ABB RobotStudio station: solution_2_AI.rspag

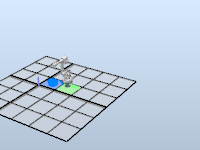
--- station ---
Station test (saved by RobotStudio 20.4.9280.0)
Controller Controller_IRB2600_12_165_C, task T_ROB1: task frame (RAPID world) sits at (1280, 730, 300) mm, rotated rx 0 ry 0 rz -90 deg in the station
Controller Controller_IRB2600_12_165_C
  mechanical unit ROB_1: IRB2600_12_165_C_01_2, 6 joints, base frame (0, 0, 0) mm
Layout (positions relative to the parent item):
  - 机器人区 [part] at (1507.5, 502.5, 0) mm
  - 方块产生区 [part]
  - 删行控制器 [smart component]
      signals: DI Rows_Delete
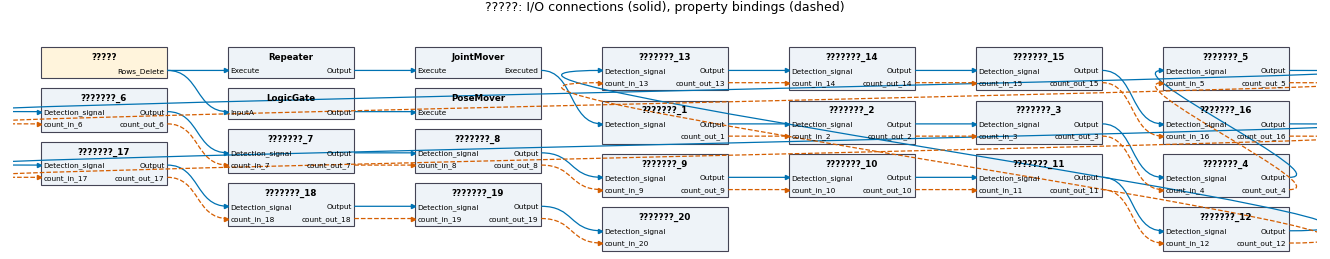
      connections:
        Repeater.Output -> JointMover.Execute
        删行控制器.Rows_Delete -> Repeater.Execute
        删行控制器.Rows_Delete -> LogicGate.InputA
        LogicGate.Output -> PoseMover.Execute
        JointMover.Executed -> 满行检测与下坠_1.Detection_signal
        满行检测与下坠_1.Output -> 满行检测与下坠_2.Detection_signal
        满行检测与下坠_2.Output -> 满行检测与下坠_3.Detection_signal
        满行检测与下坠_3.Output -> 满行检测与下坠_4.Detection_signal
        满行检测与下坠_4.Output -> 满行检测与下坠_5.Detection_signal
        满行检测与下坠_5.Output -> 满行检测与下坠_6.Detection_signal
        满行检测与下坠_6.Output -> 满行检测与下坠_7.Detection_signal
        满行检测与下坠_7.Output -> 满行检测与下坠_8.Detection_signal
        满行检测与下坠_10.Output -> 满行检测与下坠_11.Detection_signal
        满行检测与下坠_11.Output -> 满行检测与下坠_12.Detection_signal
        满行检测与下坠_12.Output -> 满行检测与下坠_13.Detection_signal
        满行检测与下坠_13.Output -> 满行检测与下坠_14.Detection_signal
        满行检测与下坠_14.Output -> 满行检测与下坠_15.Detection_signal
        满行检测与下坠_15.Output -> 满行检测与下坠_16.Detection_signal
        满行检测与下坠_16.Output -> 满行检测与下坠_17.Detection_signal
        满行检测与下坠_17.Output -> 满行检测与下坠_18.Detection_signal
        满行检测与下坠_18.Output -> 满行检测与下坠_19.Detection_signal
        满行检测与下坠_19.Output -> 满行检测与下坠_20.Detection_signal
        满行检测与下坠_8.Output -> 满行检测与下坠_9.Detection_signal
        满行检测与下坠_9.Output -> 满行检测与下坠_10.Detection_signal
        满行检测与下坠_1.count_out_1 => 满行检测与下坠_2.count_in_2
        满行检测与下坠_2.count_out_2 => 满行检测与下坠_3.count_in_3
        满行检测与下坠_3.count_out_3 => 满行检测与下坠_4.count_in_4
        满行检测与下坠_4.count_out_4 => 满行检测与下坠_5.count_in_5
        满行检测与下坠_5.count_out_5 => 满行检测与下坠_6.count_in_6
        满行检测与下坠_6.count_out_6 => 满行检测与下坠_7.count_in_7
        满行检测与下坠_7.count_out_7 => 满行检测与下坠_8.count_in_8
        满行检测与下坠_8.count_out_8 => 满行检测与下坠_9.count_in_9
        满行检测与下坠_9.count_out_9 => 满行检测与下坠_10.count_in_10
        满行检测与下坠_10.count_out_10 => 满行检测与下坠_11.count_in_11
        满行检测与下坠_11.count_out_11 => 满行检测与下坠_12.count_in_12
        满行检测与下坠_12.count_out_12 => 满行检测与下坠_13.count_in_13
        满行检测与下坠_13.count_out_13 => 满行检测与下坠_14.count_in_14
        满行检测与下坠_14.count_out_14 => 满行检测与下坠_15.count_in_15
        满行检测与下坠_15.count_out_15 => 满行检测与下坠_16.count_in_16
        满行检测与下坠_16.count_out_16 => 满行检测与下坠_17.count_in_17
        满行检测与下坠_17.count_out_17 => 满行检测与下坠_18.count_in_18
        满行检测与下坠_18.count_out_18 => 满行检测与下坠_19.count_in_19
        满行检测与下坠_19.count_out_19 => 满行检测与下坠_20.count_in_20
    - 扫描式传感器 [mechanism] at (0, -50, 0) mm; joint values [0] (rad or m)
        links: L1, L2
    - JointMover [smart component, from Components\JointMover.rslib]
        properties: Mechanism=扫描式传感器; Relative=true; Duration=0; J1=0.1
    - Repeater [smart component, from Components\Repeater.rslib]
        properties: Count=10
    - PoseMover [smart component, from Components\PoseMover.rslib]
        properties: Mechanism=扫描式传感器; Pose=0; Duration=0
    - 满行检测与下坠_1 [smart component]
        properties: count_in_1=0; count_out_1=0
        signals: DI Detection_signal, DO Output
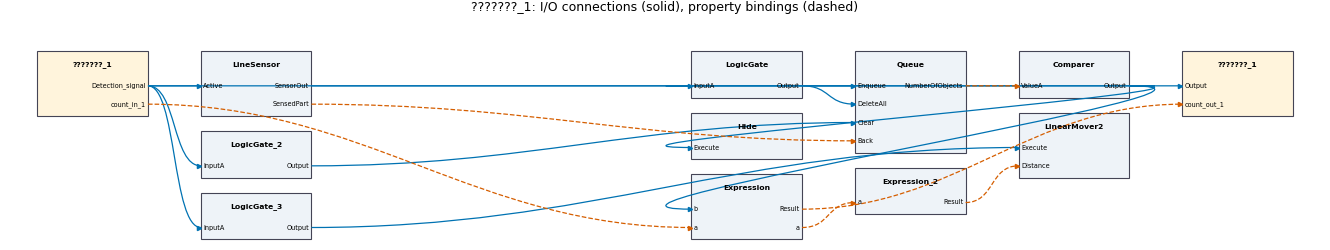
        connections:
          满行检测与下坠_1.Detection_signal -> LineSensor.Active
          LineSensor.SensorOut -> Queue.Enqueue
          Comparer.Output -> LogicGate.InputA
          LogicGate.Output -> Queue.DeleteAll
          Comparer.Output -> Hide.Execute
          LogicGate_2.Output -> Queue.Clear
          满行检测与下坠_1.Detection_signal -> LogicGate_2.InputA
          Comparer.Output -> Expression.b
          满行检测与下坠_1.Detection_signal -> LogicGate_3.InputA
          LogicGate_3.Output -> LinearMover2.Execute
          满行检测与下坠_1.Detection_signal -> 满行检测与下坠_1.Output
          LineSensor.SensedPart => Queue.Back
          Queue.NumberOfObjects => Comparer.ValueA
          满行检测与下坠_1.count_in_1 => Expression.a
          Expression.Result => 满行检测与下坠_1.count_out_1
          Expression.a => Expression_2.a
          Expression_2.Result => LinearMover2.Distance
      - LineSensor [smart component, from Components\LineSensor.rslib] at (0, 0, 40) mm
          properties: Start=[2.06 -0.045 0.01]; End=[2.13 -0.045 0.01]; Radius=0.002; SensedPart=(none); SensedPoint=[0 0 0]
        - _sensorPart_ [part]
      - Queue [smart component, from Components\Queue.rslib]
          properties: Back=(none); Front=(none); Queue=; NumberOfObjects=0
      - Comparer [smart component, from Components\Comparer.rslib]
          properties: ValueA=0; Operator===; ValueB=10
      - LogicGate [smart component, from Components\LogicGate.rslib]
          properties: Operator=NOP; Delay=0.6
      - Hide [smart component, from Components\Hide.rslib]
          properties: Object=Queue
      - LogicGate_2 [smart component, from Components\LogicGate.rslib]
          properties: Operator=NOP; Delay=0.7
      - Expression [smart component, from Components\Expression.rslib]
          properties: Expression=a+b; Result=0; a=0; b=0
      - LinearMover2 [smart component, from Components\LinearMover2.rslib]
          properties: Object=Queue; Direction=[0 0 -0.001]; Distance=0; Duration=0.5; Reference=Global; ReferenceObject=(none)
      - LogicGate_3 [smart component, from Components\LogicGate.rslib]
          properties: Operator=NOP; Delay=0.1
      - Expression_2 [smart component, from Components\Expression.rslib]
          properties: Expression=a/10; Result=0; a=0
    - LogicGate [smart component, from Components\LogicGate.rslib]
        properties: Operator=NOP; Delay=0.024
    - 满行检测与下坠_2 [smart component] at (0, 0, 100) mm
        properties: count_in_1=0; count_out_1=0; count_in_2=0; count_out_2=0
        signals: DI Detection_signal, DO Output
        connections:
          满行检测与下坠_2.Detection_signal -> LineSensor.Active
          LineSensor.SensorOut -> Queue.Enqueue
          Comparer.Output -> LogicGate.InputA
          LogicGate.Output -> Queue.DeleteAll
          Comparer.Output -> Hide.Execute
          LogicGate_2.Output -> Queue.Clear
          满行检测与下坠_2.Detection_signal -> LogicGate_2.InputA
          Comparer.Output -> Expression.b
          满行检测与下坠_2.Detection_signal -> LogicGate_3.InputA
          LogicGate_3.Output -> LinearMover2.Execute
          满行检测与下坠_2.Detection_signal -> 满行检测与下坠_2.Output
          LineSensor.SensedPart => Queue.Back
          Queue.NumberOfObjects => Comparer.ValueA
          Expression.a => Expression_2.a
          Expression_2.Result => LinearMover2.Distance
          满行检测与下坠_2.count_in_2 => Expression.a
          Expression.Result => 满行检测与下坠_2.count_out_2
      - LineSensor [smart component, from Components\LineSensor.rslib] at (0, 0, 40) mm
          properties: Start=[2.06 -0.045 0.01]; End=[2.13 -0.045 0.01]; Radius=0.002; SensedPart=(none); SensedPoint=[0 0 0]
        - _sensorPart_ [part]
      - Queue [smart component, from Components\Queue.rslib]
          properties: Back=(none); Front=(none); Queue=; NumberOfObjects=0
      - Comparer [smart component, from Components\Comparer.rslib]
          properties: ValueA=0; Operator===; ValueB=10
      - LogicGate [smart component, from Components\LogicGate.rslib]
          properties: Operator=NOP; Delay=0.6
      - Hide [smart component, from Components\Hide.rslib]
          properties: Object=Queue
      - LogicGate_2 [smart component, from Components\LogicGate.rslib]
          properties: Operator=NOP; Delay=0.7
      - Expression [smart component, from Components\Expression.rslib]
          properties: Expression=a+b; Result=0; a=0; b=0
      - LinearMover2 [smart component, from Components\LinearMover2.rslib]
          properties: Object=Queue; Direction=[0 0 -0.001]; Distance=0; Duration=0.5; Reference=Global; ReferenceObject=(none)
      - LogicGate_3 [smart component, from Components\LogicGate.rslib]
          properties: Operator=NOP; Delay=0.1
      - Expression_2 [smart component, from Components\Expression.rslib]
          properties: Expression=a/10; Result=0; a=0
    - 满行检测与下坠_3 [smart component] at (0, 0, 200) mm
        properties: count_in_1=0; count_out_1=0; count_in_3=0; count_out_3=0
        signals: DI Detection_signal, DO Output
        connections:
          满行检测与下坠_3.Detection_signal -> LineSensor.Active
          LineSensor.SensorOut -> Queue.Enqueue
          Comparer.Output -> LogicGate.InputA
          LogicGate.Output -> Queue.DeleteAll
          Comparer.Output -> Hide.Execute
          LogicGate_2.Output -> Queue.Clear
          满行检测与下坠_3.Detection_signal -> LogicGate_2.InputA
          Comparer.Output -> Expression.b
          满行检测与下坠_3.Detection_signal -> LogicGate_3.InputA
          LogicGate_3.Output -> LinearMover2.Execute
          满行检测与下坠_3.Detection_signal -> 满行检测与下坠_3.Output
          LineSensor.SensedPart => Queue.Back
          Queue.NumberOfObjects => Comparer.ValueA
          Expression.a => Expression_2.a
          Expression_2.Result => LinearMover2.Distance
          满行检测与下坠_3.count_in_3 => Expression.a
          Expression.Result => 满行检测与下坠_3.count_out_3
      - LineSensor [smart component, from Components\LineSensor.rslib] at (0, 0, 40) mm
          properties: Start=[2.06 -0.045 0.01]; End=[2.13 -0.045 0.01]; Radius=0.002; SensedPart=(none); SensedPoint=[0 0 0]
        - _sensorPart_ [part]
      - Queue [smart component, from Components\Queue.rslib]
          properties: Back=(none); Front=(none); Queue=; NumberOfObjects=0
      - Comparer [smart component, from Components\Comparer.rslib]
          properties: ValueA=0; Operator===; ValueB=10
      - LogicGate [smart component, from Components\LogicGate.rslib]
          properties: Operator=NOP; Delay=0.6
      - Hide [smart component, from Components\Hide.rslib]
          properties: Object=Queue
      - LogicGate_2 [smart component, from Components\LogicGate.rslib]
          properties: Operator=NOP; Delay=0.7
      - Expression [smart component, from Components\Expression.rslib]
          properties: Expression=a+b; Result=0; a=0; b=0
      - LinearMover2 [smart component, from Components\LinearMover2.rslib]
          properties: Object=Queue; Direction=[0 0 -0.001]; Distance=0; Duration=0.5; Reference=Global; ReferenceObject=(none)
      - LogicGate_3 [smart component, from Components\LogicGate.rslib]
          properties: Operator=NOP; Delay=0.1
      - Expression_2 [smart component, from Components\Expression.rslib]
          properties: Expression=a/10; Result=0; a=0
    - 满行检测与下坠_4 [smart component] at (0, 0, 300) mm
        properties: count_in_1=0; count_out_1=0; count_in_4=0; count_out_4=0
        signals: DI Detection_signal, DO Output
        connections:
          满行检测与下坠_4.Detection_signal -> LineSensor.Active
          LineSensor.SensorOut -> Queue.Enqueue
          Comparer.Output -> LogicGate.InputA
          LogicGate.Output -> Queue.DeleteAll
          Comparer.Output -> Hide.Execute
          LogicGate_2.Output -> Queue.Clear
          满行检测与下坠_4.Detection_signal -> LogicGate_2.InputA
          Comparer.Output -> Expression.b
          满行检测与下坠_4.Detection_signal -> LogicGate_3.InputA
          LogicGate_3.Output -> LinearMover2.Execute
          满行检测与下坠_4.Detection_signal -> 满行检测与下坠_4.Output
          LineSensor.SensedPart => Queue.Back
          Queue.NumberOfObjects => Comparer.ValueA
          Expression.a => Expression_2.a
          Expression_2.Result => LinearMover2.Distance
          满行检测与下坠_4.count_in_4 => Expression.a
          Expression.Result => 满行检测与下坠_4.count_out_4
      - LineSensor [smart component, from Components\LineSensor.rslib] at (0, 0, 40) mm
          properties: Start=[2.06 -0.045 0.01]; End=[2.13 -0.045 0.01]; Radius=0.002; SensedPart=(none); SensedPoint=[0 0 0]
        - _sensorPart_ [part]
      - Queue [smart component, from Components\Queue.rslib]
          properties: Back=(none); Front=(none); Queue=; NumberOfObjects=0
      - Comparer [smart component, from Components\Comparer.rslib]
          properties: ValueA=0; Operator===; ValueB=10
      - LogicGate [smart component, from Components\LogicGate.rslib]
          properties: Operator=NOP; Delay=0.6
      - Hide [smart component, from Components\Hide.rslib]
          properties: Object=Queue
      - LogicGate_2 [smart component, from Components\LogicGate.rslib]
          properties: Operator=NOP; Delay=0.7
      - Expression [smart component, from Components\Expression.rslib]
          properties: Expression=a+b; Result=0; a=0; b=0
      - LinearMover2 [smart component, from Components\LinearMover2.rslib]
          properties: Object=Queue; Direction=[0 0 -0.001]; Distance=0; Duration=0.5; Reference=Global; ReferenceObject=(none)
      - LogicGate_3 [smart component, from Components\LogicGate.rslib]
          properties: Operator=NOP; Delay=0.1
      - Expression_2 [smart component, from Components\Expression.rslib]
          properties: Expression=a/10; Result=0; a=0
    - 满行检测与下坠_5 [smart component] at (0, 0, 400) mm
        properties: count_in_1=0; count_out_1=0; count_in_5=0; count_out_5=0
        signals: DI Detection_signal, DO Output
        connections:
          满行检测与下坠_5.Detection_signal -> LineSensor.Active
          LineSensor.SensorOut -> Queue.Enqueue
          Comparer.Output -> LogicGate.InputA
          LogicGate.Output -> Queue.DeleteAll
          Comparer.Output -> Hide.Execute
          LogicGate_2.Output -> Queue.Clear
          满行检测与下坠_5.Detection_signal -> LogicGate_2.InputA
          Comparer.Output -> Expression.b
          满行检测与下坠_5.Detection_signal -> LogicGate_3.InputA
          LogicGate_3.Output -> LinearMover2.Execute
          满行检测与下坠_5.Detection_signal -> 满行检测与下坠_5.Output
          LineSensor.SensedPart => Queue.Back
          Queue.NumberOfObjects => Comparer.ValueA
          Expression.a => Expression_2.a
          Expression_2.Result => LinearMover2.Distance
          满行检测与下坠_5.count_in_5 => Expression.a
          Expression.Result => 满行检测与下坠_5.count_out_5
      - LineSensor [smart component, from Components\LineSensor.rslib] at (0, 0, 40) mm
          properties: Start=[2.06 -0.045 0.01]; End=[2.13 -0.045 0.01]; Radius=0.002; SensedPart=(none); SensedPoint=[0 0 0]
        - _sensorPart_ [part]
      - Queue [smart component, from Components\Queue.rslib]
          properties: Back=(none); Front=(none); Queue=; NumberOfObjects=0
      - Comparer [smart component, from Components\Comparer.rslib]
          properties: ValueA=0; Operator===; ValueB=10
      - LogicGate [smart component, from Components\LogicGate.rslib]
          properties: Operator=NOP; Delay=0.6
      - Hide [smart component, from Components\Hide.rslib]
          properties: Object=Queue
      - LogicGate_2 [smart component, from Components\LogicGate.rslib]
          properties: Operator=NOP; Delay=0.7
      - Expression [smart component, from Components\Expression.rslib]
          properties: Expression=a+b; Result=0; a=0; b=0
      - LinearMover2 [smart component, from Components\LinearMover2.rslib]
          properties: Object=Queue; Direction=[0 0 -0.001]; Distance=0; Duration=0.5; Reference=Global; ReferenceObject=(none)
      - LogicGate_3 [smart component, from Components\LogicGate.rslib]
          properties: Operator=NOP; Delay=0.1
      - Expression_2 [smart component, from Components\Expression.rslib]
          properties: Expression=a/10; Result=0; a=0
    - 满行检测与下坠_6 [smart component] at (0, 0, 500) mm
        properties: count_in_1=0; count_out_1=0; count_in_6=0; count_out_6=0
        signals: DI Detection_signal, DO Output
        connections:
          满行检测与下坠_6.Detection_signal -> LineSensor.Active
          LineSensor.SensorOut -> Queue.Enqueue
          Comparer.Output -> LogicGate.InputA
          LogicGate.Output -> Queue.DeleteAll
          Comparer.Output -> Hide.Execute
          LogicGate_2.Output -> Queue.Clear
          满行检测与下坠_6.Detection_signal -> LogicGate_2.InputA
          Comparer.Output -> Expression.b
          满行检测与下坠_6.Detection_signal -> LogicGate_3.InputA
          LogicGate_3.Output -> LinearMover2.Execute
          满行检测与下坠_6.Detection_signal -> 满行检测与下坠_6.Output
          LineSensor.SensedPart => Queue.Back
          Queue.NumberOfObjects => Comparer.ValueA
          Expression.a => Expression_2.a
          Expression_2.Result => LinearMover2.Distance
          满行检测与下坠_6.count_in_6 => Expression.a
          Expression.Result => 满行检测与下坠_6.count_out_6
      - LineSensor [smart component, from Components\LineSensor.rslib] at (0, 0, 40) mm
          properties: Start=[2.06 -0.045 0.01]; End=[2.13 -0.045 0.01]; Radius=0.002; SensedPart=(none); SensedPoint=[0 0 0]
        - _sensorPart_ [part]
      - Queue [smart component, from Components\Queue.rslib]
          properties: Back=(none); Front=(none); Queue=; NumberOfObjects=0
      - Comparer [smart component, from Components\Comparer.rslib]
          properties: ValueA=0; Operator===; ValueB=10
      - LogicGate [smart component, from Components\LogicGate.rslib]
          properties: Operator=NOP; Delay=0.6
      - Hide [smart component, from Components\Hide.rslib]
          properties: Object=Queue
      - LogicGate_2 [smart component, from Components\LogicGate.rslib]
          properties: Operator=NOP; Delay=0.7
      - Expression [smart component, from Components\Expression.rslib]
          properties: Expression=a+b; Result=0; a=0; b=0
      - LinearMover2 [smart component, from Components\LinearMover2.rslib]
          properties: Object=Queue; Direction=[0 0 -0.001]; Distance=0; Duration=0.5; Reference=Global; ReferenceObject=(none)
      - LogicGate_3 [smart component, from Components\LogicGate.rslib]
          properties: Operator=NOP; Delay=0.1
      - Expression_2 [smart component, from Components\Expression.rslib]
          properties: Expression=a/10; Result=0; a=0
    - 满行检测与下坠_7 [smart component] at (0, 0, 600) mm
        properties: count_in_1=0; count_out_1=0; count_in_7=0; count_out_8=0; count_out_7=0
        signals: DI Detection_signal, DO Output
        connections:
          满行检测与下坠_7.Detection_signal -> LineSensor.Active
          LineSensor.SensorOut -> Queue.Enqueue
          Comparer.Output -> LogicGate.InputA
          LogicGate.Output -> Queue.DeleteAll
          Comparer.Output -> Hide.Execute
          LogicGate_2.Output -> Queue.Clear
          满行检测与下坠_7.Detection_signal -> LogicGate_2.InputA
          Comparer.Output -> Expression.b
          满行检测与下坠_7.Detection_signal -> LogicGate_3.InputA
          LogicGate_3.Output -> LinearMover2.Execute
          满行检测与下坠_7.Detection_signal -> 满行检测与下坠_7.Output
          LineSensor.SensedPart => Queue.Back
          Queue.NumberOfObjects => Comparer.ValueA
          Expression.a => Expression_2.a
          Expression_2.Result => LinearMover2.Distance
          满行检测与下坠_7.count_in_7 => Expression.a
          Expression.Result => 满行检测与下坠_7.count_out_7
      - LineSensor [smart component, from Components\LineSensor.rslib] at (0, 0, 40) mm
          properties: Start=[2.06 -0.045 0.01]; End=[2.13 -0.045 0.01]; Radius=0.002; SensedPart=(none); SensedPoint=[0 0 0]
        - _sensorPart_ [part]
      - Queue [smart component, from Components\Queue.rslib]
          properties: Back=(none); Front=(none); Queue=; NumberOfObjects=0
      - Comparer [smart component, from Components\Comparer.rslib]
          properties: ValueA=0; Operator===; ValueB=10
      - LogicGate [smart component, from Components\LogicGate.rslib]
          properties: Operator=NOP; Delay=0.6
      - Hide [smart component, from Components\Hide.rslib]
          properties: Object=Queue
      - LogicGate_2 [smart component, from Components\LogicGate.rslib]
          properties: Operator=NOP; Delay=0.7
      - Expression [smart component, from Components\Expression.rslib]
          properties: Expression=a+b; Result=0; a=0; b=0
      - LinearMover2 [smart component, from Components\LinearMover2.rslib]
          properties: Object=Queue; Direction=[0 0 -0.001]; Distance=0; Duration=0.5; Reference=Global; ReferenceObject=(none)
      - LogicGate_3 [smart component, from Components\LogicGate.rslib]
          properties: Operator=NOP; Delay=0.1
      - Expression_2 [smart component, from Components\Expression.rslib]
          properties: Expression=a/10; Result=0; a=0
    - 满行检测与下坠_8 [smart component] at (0, 0, 700) mm
        properties: count_in_1=0; count_out_1=0; count_in_8=0; count_out_8=0
        signals: DI Detection_signal, DO Output
        connections:
          满行检测与下坠_8.Detection_signal -> LineSensor.Active
          LineSensor.SensorOut -> Queue.Enqueue
          Comparer.Output -> LogicGate.InputA
          LogicGate.Output -> Queue.DeleteAll
          Comparer.Output -> Hide.Execute
          LogicGate_2.Output -> Queue.Clear
          满行检测与下坠_8.Detection_signal -> LogicGate_2.InputA
          Comparer.Output -> Expression.b
          满行检测与下坠_8.Detection_signal -> LogicGate_3.InputA
          LogicGate_3.Output -> LinearMover2.Execute
          满行检测与下坠_8.Detection_signal -> 满行检测与下坠_8.Output
          LineSensor.SensedPart => Queue.Back
          Queue.NumberOfObjects => Comparer.ValueA
          Expression.a => Expression_2.a
          Expression_2.Result => LinearMover2.Distance
          满行检测与下坠_8.count_in_8 => Expression.a
          Expression.Result => 满行检测与下坠_8.count_out_8
      - LineSensor [smart component, from Components\LineSensor.rslib] at (0, 0, 40) mm
          properties: Start=[2.06 -0.045 0.01]; End=[2.13 -0.045 0.01]; Radius=0.002; SensedPart=(none); SensedPoint=[0 0 0]
        - _sensorPart_ [part]
      - Queue [smart component, from Components\Queue.rslib]
          properties: Back=(none); Front=(none); Queue=; NumberOfObjects=0
      - Comparer [smart component, from Components\Comparer.rslib]
          properties: ValueA=0; Operator===; ValueB=10
      - LogicGate [smart component, from Components\LogicGate.rslib]
          properties: Operator=NOP; Delay=0.6
      - Hide [smart component, from Components\Hide.rslib]
          properties: Object=Queue
      - LogicGate_2 [smart component, from Components\LogicGate.rslib]
          properties: Operator=NOP; Delay=0.7
      - Expression [smart component, from Components\Expression.rslib]
          properties: Expression=a+b; Result=0; a=0; b=0
      - LinearMover2 [smart component, from Components\LinearMover2.rslib]
          properties: Object=Queue; Direction=[0 0 -0.001]; Distance=0; Duration=0.5; Reference=Global; ReferenceObject=(none)
      - LogicGate_3 [smart component, from Components\LogicGate.rslib]
          properties: Operator=NOP; Delay=0.1
      - Expression_2 [smart component, from Components\Expression.rslib]
          properties: Expression=a/10; Result=0; a=0
    - 满行检测与下坠_9 [smart component] at (0, 0, 800) mm
        properties: count_in_1=0; count_out_1=0; count_in_9=0; count_out_9=0
        signals: DI Detection_signal, DO Output
        connections:
          满行检测与下坠_9.Detection_signal -> LineSensor.Active
          LineSensor.SensorOut -> Queue.Enqueue
          Comparer.Output -> LogicGate.InputA
          LogicGate.Output -> Queue.DeleteAll
          Comparer.Output -> Hide.Execute
          LogicGate_2.Output -> Queue.Clear
          满行检测与下坠_9.Detection_signal -> LogicGate_2.InputA
          Comparer.Output -> Expression.b
          满行检测与下坠_9.Detection_signal -> LogicGate_3.InputA
          LogicGate_3.Output -> LinearMover2.Execute
          满行检测与下坠_9.Detection_signal -> 满行检测与下坠_9.Output
          LineSensor.SensedPart => Queue.Back
          Queue.NumberOfObjects => Comparer.ValueA
          Expression.a => Expression_2.a
          Expression_2.Result => LinearMover2.Distance
          满行检测与下坠_9.count_in_9 => Expression.a
          Expression.Result => 满行检测与下坠_9.count_out_9
      - LineSensor [smart component, from Components\LineSensor.rslib] at (0, 0, 40) mm
          properties: Start=[2.06 -0.045 0.01]; End=[2.13 -0.045 0.01]; Radius=0.002; SensedPart=(none); SensedPoint=[0 0 0]
        - _sensorPart_ [part]
      - Queue [smart component, from Components\Queue.rslib]
          properties: Back=(none); Front=(none); Queue=; NumberOfObjects=0
      - Comparer [smart component, from Components\Comparer.rslib]
          properties: ValueA=0; Operator===; ValueB=10
      - LogicGate [smart component, from Components\LogicGate.rslib]
          properties: Operator=NOP; Delay=0.6
      - Hide [smart component, from Components\Hide.rslib]
          properties: Object=Queue
      - LogicGate_2 [smart component, from Components\LogicGate.rslib]
          properties: Operator=NOP; Delay=0.7
      - Expression [smart component, from Components\Expression.rslib]
          properties: Expression=a+b; Result=0; a=0; b=0
      - LinearMover2 [smart component, from Components\LinearMover2.rslib]
          properties: Object=Queue; Direction=[0 0 -0.001]; Distance=0; Duration=0.5; Reference=Global; ReferenceObject=(none)
      - LogicGate_3 [smart component, from Components\LogicGate.rslib]
          properties: Operator=NOP; Delay=0.1
      - Expression_2 [smart component, from Components\Expression.rslib]
          properties: Expression=a/10; Result=0; a=0
    - 满行检测与下坠_10 [smart component] at (0, 0, 900) mm
        properties: count_in_1=0; count_out_1=0; count_out_10=0; count_in_10=0
        signals: DI Detection_signal, DO Output
        connections:
          满行检测与下坠_10.Detection_signal -> LineSensor.Active
          LineSensor.SensorOut -> Queue.Enqueue
          Comparer.Output -> LogicGate.InputA
          LogicGate.Output -> Queue.DeleteAll
          Comparer.Output -> Hide.Execute
          LogicGate_2.Output -> Queue.Clear
          满行检测与下坠_10.Detection_signal -> LogicGate_2.InputA
          Comparer.Output -> Expression.b
          满行检测与下坠_10.Detection_signal -> LogicGate_3.InputA
          LogicGate_3.Output -> LinearMover2.Execute
          满行检测与下坠_10.Detection_signal -> 满行检测与下坠_10.Output
          LineSensor.SensedPart => Queue.Back
          Queue.NumberOfObjects => Comparer.ValueA
          Expression.a => Expression_2.a
          Expression_2.Result => LinearMover2.Distance
          满行检测与下坠_10.count_in_10 => Expression.a
          Expression.Result => 满行检测与下坠_10.count_out_10
      - LineSensor [smart component, from Components\LineSensor.rslib] at (0, 0, 40) mm
          properties: Start=[2.06 -0.045 0.01]; End=[2.13 -0.045 0.01]; Radius=0.002; SensedPart=(none); SensedPoint=[0 0 0]
        - _sensorPart_ [part]
      - Queue [smart component, from Components\Queue.rslib]
          properties: Back=(none); Front=(none); Queue=; NumberOfObjects=0
      - Comparer [smart component, from Components\Comparer.rslib]
          properties: ValueA=0; Operator===; ValueB=10
      - LogicGate [smart component, from Components\LogicGate.rslib]
          properties: Operator=NOP; Delay=0.6
      - Hide [smart component, from Components\Hide.rslib]
          properties: Object=Queue
      - LogicGate_2 [smart component, from Components\LogicGate.rslib]
          properties: Operator=NOP; Delay=0.7
      - Expression [smart component, from Components\Expression.rslib]
          properties: Expression=a+b; Result=0; a=0; b=0
      - LinearMover2 [smart component, from Components\LinearMover2.rslib]
          properties: Object=Queue; Direction=[0 0 -0.001]; Distance=0; Duration=0.5; Reference=Global; ReferenceObject=(none)
      - LogicGate_3 [smart component, from Components\LogicGate.rslib]
          properties: Operator=NOP; Delay=0.1
      - Expression_2 [smart component, from Components\Expression.rslib]
          properties: Expression=a/10; Result=0; a=0
    - 满行检测与下坠_11 [smart component] at (0, 0, 1000) mm
        properties: count_in_1=0; count_out_1=0; count_out_11=0; count_in_11=0
        signals: DI Detection_signal, DO Output
        connections:
          满行检测与下坠_11.Detection_signal -> LineSensor.Active
          LineSensor.SensorOut -> Queue.Enqueue
          Comparer.Output -> LogicGate.InputA
          LogicGate.Output -> Queue.DeleteAll
          Comparer.Output -> Hide.Execute
          LogicGate_2.Output -> Queue.Clear
          满行检测与下坠_11.Detection_signal -> LogicGate_2.InputA
          Comparer.Output -> Expression.b
          满行检测与下坠_11.Detection_signal -> LogicGate_3.InputA
          LogicGate_3.Output -> LinearMover2.Execute
          满行检测与下坠_11.Detection_signal -> 满行检测与下坠_11.Output
          LineSensor.SensedPart => Queue.Back
          Queue.NumberOfObjects => Comparer.ValueA
          Expression.a => Expression_2.a
          Expression_2.Result => LinearMover2.Distance
          满行检测与下坠_11.count_in_11 => Expression.a
          Expression.Result => 满行检测与下坠_11.count_out_11
      - LineSensor [smart component, from Components\LineSensor.rslib] at (0, 0, 40) mm
          properties: Start=[2.06 -0.045 0.01]; End=[2.13 -0.045 0.01]; Radius=0.002; SensedPart=(none); SensedPoint=[0 0 0]
        - _sensorPart_ [part]
      - Queue [smart component, from Components\Queue.rslib]
          properties: Back=(none); Front=(none); Queue=; NumberOfObjects=0
      - Comparer [smart component, from Components\Comparer.rslib]
          properties: ValueA=0; Operator===; ValueB=10
      - LogicGate [smart component, from Components\LogicGate.rslib]
          properties: Operator=NOP; Delay=0.6
      - Hide [smart component, from Components\Hide.rslib]
          properties: Object=Queue
      - LogicGate_2 [smart component, from Components\LogicGate.rslib]
          properties: Operator=NOP; Delay=0.7
      - Expression [smart component, from Components\Expression.rslib]
          properties: Expression=a+b; Result=0; a=0; b=0
      - LinearMover2 [smart component, from Components\LinearMover2.rslib]
          properties: Object=Queue; Direction=[0 0 -0.001]; Distance=0; Duration=0.5; Reference=Global; ReferenceObject=(none)
      - LogicGate_3 [smart component, from Components\LogicGate.rslib]
          properties: Operator=NOP; Delay=0.1
      - Expression_2 [smart component, from Components\Expression.rslib]
          properties: Expression=a/10; Result=0; a=0
    - 满行检测与下坠_12 [smart component] at (0, 0, 1100) mm
        properties: count_in_1=0; count_out_1=0; count_out_12=0; count_in_12=0
        signals: DI Detection_signal, DO Output
        connections:
          满行检测与下坠_12.Detection_signal -> LineSensor.Active
          LineSensor.SensorOut -> Queue.Enqueue
          Comparer.Output -> LogicGate.InputA
          LogicGate.Output -> Queue.DeleteAll
          Comparer.Output -> Hide.Execute
          LogicGate_2.Output -> Queue.Clear
          满行检测与下坠_12.Detection_signal -> LogicGate_2.InputA
          Comparer.Output -> Expression.b
          满行检测与下坠_12.Detection_signal -> LogicGate_3.InputA
          LogicGate_3.Output -> LinearMover2.Execute
          满行检测与下坠_12.Detection_signal -> 满行检测与下坠_12.Output
          LineSensor.SensedPart => Queue.Back
          Queue.NumberOfObjects => Comparer.ValueA
          Expression.a => Expression_2.a
          Expression_2.Result => LinearMover2.Distance
          满行检测与下坠_12.count_in_12 => Expression.a
          Expression.Result => 满行检测与下坠_12.count_out_12
      - LineSensor [smart component, from Components\LineSensor.rslib] at (0, 0, 40) mm
          properties: Start=[2.06 -0.045 0.01]; End=[2.13 -0.045 0.01]; Radius=0.002; SensedPart=(none); SensedPoint=[0 0 0]
        - _sensorPart_ [part]
      - Queue [smart component, from Components\Queue.rslib]
          properties: Back=(none); Front=(none); Queue=; NumberOfObjects=0
      - Comparer [smart component, from Components\Comparer.rslib]
          properties: ValueA=0; Operator===; ValueB=10
      - LogicGate [smart component, from Components\LogicGate.rslib]
          properties: Operator=NOP; Delay=0.6
      - Hide [smart component, from Components\Hide.rslib]
          properties: Object=Queue
      - LogicGate_2 [smart component, from Components\LogicGate.rslib]
          properties: Operator=NOP; Delay=0.7
      - Expression [smart component, from Components\Expression.rslib]
          properties: Expression=a+b; Result=0; a=0; b=0
      - LinearMover2 [smart component, from Components\LinearMover2.rslib]
          properties: Object=Queue; Direction=[0 0 -0.001]; Distance=0; Duration=0.5; Reference=Global; ReferenceObject=(none)
      - LogicGate_3 [smart component, from Components\LogicGate.rslib]
          properties: Operator=NOP; Delay=0.1
      - Expression_2 [smart component, from Components\Expression.rslib]
          properties: Expression=a/10; Result=0; a=0
    - 满行检测与下坠_13 [smart component] at (0, 0, 1200) mm
        properties: count_in_1=0; count_out_1=0; count_out_13=0; count_in_13=0
        signals: DI Detection_signal, DO Output
        connections:
          满行检测与下坠_13.Detection_signal -> LineSensor.Active
          LineSensor.SensorOut -> Queue.Enqueue
          Comparer.Output -> LogicGate.InputA
          LogicGate.Output -> Queue.DeleteAll
          Comparer.Output -> Hide.Execute
          LogicGate_2.Output -> Queue.Clear
          满行检测与下坠_13.Detection_signal -> LogicGate_2.InputA
          Comparer.Output -> Expression.b
          满行检测与下坠_13.Detection_signal -> LogicGate_3.InputA
          LogicGate_3.Output -> LinearMover2.Execute
          满行检测与下坠_13.Detection_signal -> 满行检测与下坠_13.Output
          LineSensor.SensedPart => Queue.Back
          Queue.NumberOfObjects => Comparer.ValueA
          Expression.a => Expression_2.a
          Expression_2.Result => LinearMover2.Distance
          满行检测与下坠_13.count_in_13 => Expression.a
          Expression.Result => 满行检测与下坠_13.count_out_13
      - LineSensor [smart component, from Components\LineSensor.rslib] at (0, 0, 40) mm
          properties: Start=[2.06 -0.045 0.01]; End=[2.13 -0.045 0.01]; Radius=0.002; SensedPart=(none); SensedPoint=[0 0 0]
        - _sensorPart_ [part]
      - Queue [smart component, from Components\Queue.rslib]
          properties: Back=(none); Front=(none); Queue=; NumberOfObjects=0
      - Comparer [smart component, from Components\Comparer.rslib]
          properties: ValueA=0; Operator===; ValueB=10
      - LogicGate [smart component, from Components\LogicGate.rslib]
          properties: Operator=NOP; Delay=0.6
      - Hide [smart component, from Components\Hide.rslib]
          properties: Object=Queue
      - LogicGate_2 [smart component, from Components\LogicGate.rslib]
          properties: Operator=NOP; Delay=0.7
      - Expression [smart component, from Components\Expression.rslib]
          properties: Expression=a+b; Result=0; a=0; b=0
      - LinearMover2 [smart component, from Components\LinearMover2.rslib]
          properties: Object=Queue; Direction=[0 0 -0.001]; Distance=0; Duration=0.5; Reference=Global; ReferenceObject=(none)
      - LogicGate_3 [smart component, from Components\LogicGate.rslib]
          properties: Operator=NOP; Delay=0.1
      - Expression_2 [smart component, from Components\Expression.rslib]
          properties: Expression=a/10; Result=0; a=0
    - 满行检测与下坠_14 [smart component] at (0, 0, 1300) mm
        properties: count_in_1=0; count_out_1=0; count_out_14=0; count_in_14=0
        signals: DI Detection_signal, DO Output
        connections:
          满行检测与下坠_14.Detection_signal -> LineSensor.Active
          LineSensor.SensorOut -> Queue.Enqueue
          Comparer.Output -> LogicGate.InputA
          LogicGate.Output -> Queue.DeleteAll
          Comparer.Output -> Hide.Execute
          LogicGate_2.Output -> Queue.Clear
          满行检测与下坠_14.Detection_signal -> LogicGate_2.InputA
          Comparer.Output -> Expression.b
          满行检测与下坠_14.Detection_signal -> LogicGate_3.InputA
          LogicGate_3.Output -> LinearMover2.Execute
          满行检测与下坠_14.Detection_signal -> 满行检测与下坠_14.Output
          LineSensor.SensedPart => Queue.Back
          Queue.NumberOfObjects => Comparer.ValueA
          Expression.a => Expression_2.a
          Expression_2.Result => LinearMover2.Distance
          满行检测与下坠_14.count_in_14 => Expression.a
          Expression.Result => 满行检测与下坠_14.count_out_14
      - LineSensor [smart component, from Components\LineSensor.rslib] at (0, 0, 40) mm
          properties: Start=[2.06 -0.045 0.01]; End=[2.13 -0.045 0.01]; Radius=0.002; SensedPart=(none); SensedPoint=[0 0 0]
        - _sensorPart_ [part]
      - Queue [smart component, from Components\Queue.rslib]
          properties: Back=(none); Front=(none); Queue=; NumberOfObjects=0
      - Comparer [smart component, from Components\Comparer.rslib]
          properties: ValueA=0; Operator===; ValueB=10
      - LogicGate [smart component, from Components\LogicGate.rslib]
          properties: Operator=NOP; Delay=0.6
      - Hide [smart component, from Components\Hide.rslib]
          properties: Object=Queue
      - LogicGate_2 [smart component, from Components\LogicGate.rslib]
          properties: Operator=NOP; Delay=0.7
      - Expression [smart component, from Components\Expression.rslib]
          properties: Expression=a+b; Result=0; a=0; b=0
      - LinearMover2 [smart component, from Components\LinearMover2.rslib]
          properties: Object=Queue; Direction=[0 0 -0.001]; Distance=0; Duration=0.5; Reference=Global; ReferenceObject=(none)
      - LogicGate_3 [smart component, from Components\LogicGate.rslib]
          properties: Operator=NOP; Delay=0.1
      - Expression_2 [smart component, from Components\Expression.rslib]
          properties: Expression=a/10; Result=0; a=0
    - 满行检测与下坠_15 [smart component] at (0, 0, 1400) mm
        properties: count_in_1=0; count_out_1=0; count_out_15=0; count_in_15=0
        signals: DI Detection_signal, DO Output
        connections:
          满行检测与下坠_15.Detection_signal -> LineSensor.Active
          LineSensor.SensorOut -> Queue.Enqueue
          Comparer.Output -> LogicGate.InputA
          LogicGate.Output -> Queue.DeleteAll
          Comparer.Output -> Hide.Execute
          LogicGate_2.Output -> Queue.Clear
          满行检测与下坠_15.Detection_signal -> LogicGate_2.InputA
          Comparer.Output -> Expression.b
          满行检测与下坠_15.Detection_signal -> LogicGate_3.InputA
          LogicGate_3.Output -> LinearMover2.Execute
          满行检测与下坠_15.Detection_signal -> 满行检测与下坠_15.Output
          LineSensor.SensedPart => Queue.Back
          Queue.NumberOfObjects => Comparer.ValueA
          Expression.a => Expression_2.a
          Expression_2.Result => LinearMover2.Distance
          满行检测与下坠_15.count_in_15 => Expression.a
          Expression.Result => 满行检测与下坠_15.count_out_15
      - LineSensor [smart component, from Components\LineSensor.rslib] at (0, 0, 40) mm
          properties: Start=[2.06 -0.045 0.01]; End=[2.13 -0.045 0.01]; Radius=0.002; SensedPart=(none); SensedPoint=[0 0 0]
        - _sensorPart_ [part]
      - Queue [smart component, from Components\Queue.rslib]
          properties: Back=(none); Front=(none); Queue=; NumberOfObjects=0
      - Comparer [smart component, from Components\Comparer.rslib]
          properties: ValueA=0; Operator===; ValueB=10
      - LogicGate [smart component, from Components\LogicGate.rslib]
          properties: Operator=NOP; Delay=0.6
      - Hide [smart component, from Components\Hide.rslib]
          properties: Object=Queue
      - LogicGate_2 [smart component, from Components\LogicGate.rslib]
          properties: Operator=NOP; Delay=0.7
      - Expression [smart component, from Components\Expression.rslib]
          properties: Expression=a+b; Result=0; a=0; b=0
      - LinearMover2 [smart component, from Components\LinearMover2.rslib]
          properties: Object=Queue; Direction=[0 0 -0.001]; Distance=0; Duration=0.5; Reference=Global; ReferenceObject=(none)
      - LogicGate_3 [smart component, from Components\LogicGate.rslib]
          properties: Operator=NOP; Delay=0.1
      - Expression_2 [smart component, from Components\Expression.rslib]
          properties: Expression=a/10; Result=0; a=0
    - 满行检测与下坠_16 [smart component] at (0, 0, 1500) mm
        properties: count_in_1=0; count_out_1=0; count_out_16=0; count_in_16=0
        signals: DI Detection_signal, DO Output
        connections:
          满行检测与下坠_16.Detection_signal -> LineSensor.Active
          LineSensor.SensorOut -> Queue.Enqueue
          Comparer.Output -> LogicGate.InputA
          LogicGate.Output -> Queue.DeleteAll
          Comparer.Output -> Hide.Execute
          LogicGate_2.Output -> Queue.Clear
          满行检测与下坠_16.Detection_signal -> LogicGate_2.InputA
          Comparer.Output -> Expression.b
          满行检测与下坠_16.Detection_signal -> LogicGate_3.InputA
          LogicGate_3.Output -> LinearMover2.Execute
          满行检测与下坠_16.Detection_signal -> 满行检测与下坠_16.Output
          LineSensor.SensedPart => Queue.Back
          Queue.NumberOfObjects => Comparer.ValueA
          Expression.a => Expression_2.a
          Expression_2.Result => LinearMover2.Distance
          满行检测与下坠_16.count_in_16 => Expression.a
          Expression.Result => 满行检测与下坠_16.count_out_16
      - LineSensor [smart component, from Components\LineSensor.rslib] at (0, 0, 40) mm
          properties: Start=[2.06 -0.045 0.01]; End=[2.13 -0.045 0.01]; Radius=0.002; SensedPart=(none); SensedPoint=[0 0 0]
        - _sensorPart_ [part]
      - Queue [smart component, from Components\Queue.rslib]
          properties: Back=(none); Front=(none); Queue=; NumberOfObjects=0
      - Comparer [smart component, from Components\Comparer.rslib]
          properties: ValueA=0; Operator===; ValueB=10
      - LogicGate [smart component, from Components\LogicGate.rslib]
          properties: Operator=NOP; Delay=0.6
      - Hide [smart component, from Components\Hide.rslib]
          properties: Object=Queue
      - LogicGate_2 [smart component, from Components\LogicGate.rslib]
          properties: Operator=NOP; Delay=0.7
      - Expression [smart component, from Components\Expression.rslib]
          properties: Expression=a+b; Result=0; a=0; b=0
      - LinearMover2 [smart component, from Components\LinearMover2.rslib]
          properties: Object=Queue; Direction=[0 0 -0.001]; Distance=0; Duration=0.5; Reference=Global; ReferenceObject=(none)
      - LogicGate_3 [smart component, from Components\LogicGate.rslib]
          properties: Operator=NOP; Delay=0.1
      - Expression_2 [smart component, from Components\Expression.rslib]
          properties: Expression=a/10; Result=0; a=0
    - 满行检测与下坠_17 [smart component] at (0, 0, 1600) mm
        properties: count_in_1=0; count_out_1=0; count_out_17=0; count_in_17=0
        signals: DI Detection_signal, DO Output
        connections:
          满行检测与下坠_17.Detection_signal -> LineSensor.Active
          LineSensor.SensorOut -> Queue.Enqueue
          Comparer.Output -> LogicGate.InputA
          LogicGate.Output -> Queue.DeleteAll
          Comparer.Output -> Hide.Execute
          LogicGate_2.Output -> Queue.Clear
          满行检测与下坠_17.Detection_signal -> LogicGate_2.InputA
          Comparer.Output -> Expression.b
          满行检测与下坠_17.Detection_signal -> LogicGate_3.InputA
          LogicGate_3.Output -> LinearMover2.Execute
          满行检测与下坠_17.Detection_signal -> 满行检测与下坠_17.Output
          LineSensor.SensedPart => Queue.Back
          Queue.NumberOfObjects => Comparer.ValueA
          Expression.a => Expression_2.a
          Expression_2.Result => LinearMover2.Distance
          Expression.Result => 满行检测与下坠_17.count_out_17
          满行检测与下坠_17.count_in_17 => Expression.a
      - LineSensor [smart component, from Components\LineSensor.rslib] at (0, 0, 40) mm
          properties: Start=[2.06 -0.045 0.01]; End=[2.13 -0.045 0.01]; Radius=0.002; SensedPart=(none); SensedPoint=[0 0 0]
        - _sensorPart_ [part]
      - Queue [smart component, from Components\Queue.rslib]
          properties: Back=(none); Front=(none); Queue=; NumberOfObjects=0
      - Comparer [smart component, from Components\Comparer.rslib]
          properties: ValueA=0; Operator===; ValueB=10
      - LogicGate [smart component, from Components\LogicGate.rslib]
          properties: Operator=NOP; Delay=0.6
      - Hide [smart component, from Components\Hide.rslib]
          properties: Object=Queue
      - LogicGate_2 [smart component, from Components\LogicGate.rslib]
          properties: Operator=NOP; Delay=0.7
      - Expression [smart component, from Components\Expression.rslib]
          properties: Expression=a+b; Result=0; a=0; b=0
      - LinearMover2 [smart component, from Components\LinearMover2.rslib]
          properties: Object=Queue; Direction=[0 0 -0.001]; Distance=0; Duration=0.5; Reference=Global; ReferenceObject=(none)
      - LogicGate_3 [smart component, from Components\LogicGate.rslib]
          properties: Operator=NOP; Delay=0.1
      - Expression_2 [smart component, from Components\Expression.rslib]
          properties: Expression=a/10; Result=0; a=0
    - 满行检测与下坠_18 [smart component] at (0, 0, 1700) mm
        properties: count_in_1=0; count_out_1=0; count_out_18=0; count_in_18=0
        signals: DI Detection_signal, DO Output
        connections:
          满行检测与下坠_18.Detection_signal -> LineSensor.Active
          LineSensor.SensorOut -> Queue.Enqueue
          Comparer.Output -> LogicGate.InputA
          LogicGate.Output -> Queue.DeleteAll
          Comparer.Output -> Hide.Execute
          LogicGate_2.Output -> Queue.Clear
          满行检测与下坠_18.Detection_signal -> LogicGate_2.InputA
          Comparer.Output -> Expression.b
          满行检测与下坠_18.Detection_signal -> LogicGate_3.InputA
          LogicGate_3.Output -> LinearMover2.Execute
          满行检测与下坠_18.Detection_signal -> 满行检测与下坠_18.Output
          LineSensor.SensedPart => Queue.Back
          Queue.NumberOfObjects => Comparer.ValueA
          Expression.a => Expression_2.a
          Expression_2.Result => LinearMover2.Distance
          满行检测与下坠_18.count_in_18 => Expression.a
          Expression.Result => 满行检测与下坠_18.count_out_18
      - LineSensor [smart component, from Components\LineSensor.rslib] at (0, 0, 40) mm
          properties: Start=[2.06 -0.045 0.01]; End=[2.13 -0.045 0.01]; Radius=0.002; SensedPart=(none); SensedPoint=[0 0 0]
        - _sensorPart_ [part]
      - Queue [smart component, from Components\Queue.rslib]
          properties: Back=(none); Front=(none); Queue=; NumberOfObjects=0
      - Comparer [smart component, from Components\Comparer.rslib]
          properties: ValueA=0; Operator===; ValueB=10
      - LogicGate [smart component, from Components\LogicGate.rslib]
          properties: Operator=NOP; Delay=0.6
      - Hide [smart component, from Components\Hide.rslib]
          properties: Object=Queue
      - LogicGate_2 [smart component, from Components\LogicGate.rslib]
          properties: Operator=NOP; Delay=0.7
      - Expression [smart component, from Components\Expression.rslib]
          properties: Expression=a+b; Result=0; a=0; b=0
      - LinearMover2 [smart component, from Components\LinearMover2.rslib]
          properties: Object=Queue; Direction=[0 0 -0.001]; Distance=0; Duration=0.5; Reference=Global; ReferenceObject=(none)
      - LogicGate_3 [smart component, from Components\LogicGate.rslib]
          properties: Operator=NOP; Delay=0.1
      - Expression_2 [smart component, from Components\Expression.rslib]
          properties: Expression=a/10; Result=0; a=0
    - 满行检测与下坠_19 [smart component] at (0, 0, 1800) mm
        properties: count_in_1=0; count_out_1=0; count_out_19=0; count_in_19=0
        signals: DI Detection_signal, DO Output
        connections:
          满行检测与下坠_19.Detection_signal -> LineSensor.Active
          LineSensor.SensorOut -> Queue.Enqueue
          Comparer.Output -> LogicGate.InputA
          LogicGate.Output -> Queue.DeleteAll
          Comparer.Output -> Hide.Execute
          LogicGate_2.Output -> Queue.Clear
          满行检测与下坠_19.Detection_signal -> LogicGate_2.InputA
          Comparer.Output -> Expression.b
          满行检测与下坠_19.Detection_signal -> LogicGate_3.InputA
          LogicGate_3.Output -> LinearMover2.Execute
          满行检测与下坠_19.Detection_signal -> 满行检测与下坠_19.Output
          LineSensor.SensedPart => Queue.Back
          Queue.NumberOfObjects => Comparer.ValueA
          Expression.a => Expression_2.a
          Expression_2.Result => LinearMover2.Distance
          满行检测与下坠_19.count_in_19 => Expression.a
          Expression.Result => 满行检测与下坠_19.count_out_19
      - LineSensor [smart component, from Components\LineSensor.rslib] at (0, 0, 40) mm
          properties: Start=[2.06 -0.045 0.01]; End=[2.13 -0.045 0.01]; Radius=0.002; SensedPart=(none); SensedPoint=[0 0 0]
        - _sensorPart_ [part]
      - Queue [smart component, from Components\Queue.rslib]
          properties: Back=(none); Front=(none); Queue=; NumberOfObjects=0
      - Comparer [smart component, from Components\Comparer.rslib]
          properties: ValueA=0; Operator===; ValueB=10
      - LogicGate [smart component, from Components\LogicGate.rslib]
          properties: Operator=NOP; Delay=0.6
      - Hide [smart component, from Components\Hide.rslib]
          properties: Object=Queue
      - LogicGate_2 [smart component, from Components\LogicGate.rslib]
          properties: Operator=NOP; Delay=0.7
      - Expression [smart component, from Components\Expression.rslib]
          properties: Expression=a+b; Result=0; a=0; b=0
      - LinearMover2 [smart component, from Components\LinearMover2.rslib]
          properties: Object=Queue; Direction=[0 0 -0.001]; Distance=0; Duration=0.5; Reference=Global; ReferenceObject=(none)
      - LogicGate_3 [smart component, from Components\LogicGate.rslib]
          properties: Operator=NOP; Delay=0.1
      - Expression_2 [smart component, from Components\Expression.rslib]
          properties: Expression=a/10; Result=0; a=0
    - 满行检测与下坠_20 [smart component] at (0, 0, 1900) mm
        properties: count_in_1=0; count_out_1=0; count_out_20=0; count_in_20=0
        signals: DI Detection_signal, DO Output
        connections:
          满行检测与下坠_20.Detection_signal -> LineSensor.Active
          LineSensor.SensorOut -> Queue.Enqueue
          Comparer.Output -> LogicGate.InputA
          LogicGate.Output -> Queue.DeleteAll
          Comparer.Output -> Hide.Execute
          LogicGate_2.Output -> Queue.Clear
          满行检测与下坠_20.Detection_signal -> LogicGate_2.InputA
          Comparer.Output -> Expression.b
          满行检测与下坠_20.Detection_signal -> LogicGate_3.InputA
          LogicGate_3.Output -> LinearMover2.Execute
          满行检测与下坠_20.Detection_signal -> 满行检测与下坠_20.Output
          LineSensor.SensedPart => Queue.Back
          Queue.NumberOfObjects => Comparer.ValueA
          Expression.a => Expression_2.a
          Expression_2.Result => LinearMover2.Distance
          满行检测与下坠_20.count_in_20 => Expression.a
          Expression.Result => 满行检测与下坠_20.count_out_20
      - LineSensor [smart component, from Components\LineSensor.rslib] at (0, 0, 40) mm
          properties: Start=[2.06 -0.045 0.01]; End=[2.13 -0.045 0.01]; Radius=0.002; SensedPart=(none); SensedPoint=[0 0 0]
        - _sensorPart_ [part]
      - Queue [smart component, from Components\Queue.rslib]
          properties: Back=(none); Front=(none); Queue=; NumberOfObjects=0
      - Comparer [smart component, from Components\Comparer.rslib]
          properties: ValueA=0; Operator===; ValueB=10
      - LogicGate [smart component, from Components\LogicGate.rslib]
          properties: Operator=NOP; Delay=0.6
      - Hide [smart component, from Components\Hide.rslib]
          properties: Object=Queue
      - LogicGate_2 [smart component, from Components\LogicGate.rslib]
          properties: Operator=NOP; Delay=0.7
      - Expression [smart component, from Components\Expression.rslib]
          properties: Expression=a+b; Result=0; a=0; b=0
      - LinearMover2 [smart component, from Components\LinearMover2.rslib]
          properties: Object=Queue; Direction=[0 0 -0.001]; Distance=0; Duration=0.5; Reference=Global; ReferenceObject=(none)
      - LogicGate_3 [smart component, from Components\LogicGate.rslib]
          properties: Operator=NOP; Delay=0.1
      - Expression_2 [smart component, from Components\Expression.rslib]
          properties: Expression=a/10; Result=0; a=0
  - 20*10方块矩阵区 [smart component]
    - MatrixRepeater [smart component, from Components\MatrixRepeater.rslib]
        properties: Source=小方块（源对象）; CountX=1; CountY=10; CountZ=20; OffsetX=0.1; OffsetY=0.1; OffsetZ=0.1
      - 小方块（源对象） [part]
      - 小方块（源对象） [part] at (0, 100, 0) mm
      - 小方块（源对象） [part] at (0, 200, 0) mm
      - 小方块（源对象） [part] at (0, 300, 0) mm
      - 小方块（源对象） [part] at (0, 400, 0) mm
      - 小方块（源对象） [part] at (0, 500, 0) mm
      - 小方块（源对象） [part] at (0, 600, 0) mm
      - 小方块（源对象） [part] at (0, 700, 0) mm
      - 小方块（源对象） [part] at (0, 800, 0) mm
      - 小方块（源对象） [part] at (0, 900, 0) mm
      - 小方块（源对象） [part] at (0, 0, 100) mm
      - 小方块（源对象） [part] at (0, 100, 100) mm
      - 小方块（源对象） [part] at (0, 200, 100) mm
      - 小方块（源对象） [part] at (0, 300, 100) mm
      - 小方块（源对象） [part] at (0, 400, 100) mm
      - 小方块（源对象） [part] at (0, 500, 100) mm
      - 小方块（源对象） [part] at (0, 600, 100) mm
      - 小方块（源对象） [part] at (0, 700, 100) mm
      - 小方块（源对象） [part] at (0, 800, 100) mm
      - 小方块（源对象） [part] at (0, 900, 100) mm
      - 小方块（源对象） [part] at (0, 0, 200) mm
      - 小方块（源对象） [part] at (0, 100, 200) mm
      - 小方块（源对象） [part] at (0, 200, 200) mm
      - 小方块（源对象） [part] at (0, 300, 200) mm
      - 小方块（源对象） [part] at (0, 400, 200) mm
      - 小方块（源对象） [part] at (0, 500, 200) mm
      - 小方块（源对象） [part] at (0, 600, 200) mm
      - 小方块（源对象） [part] at (0, 700, 200) mm
      - 小方块（源对象） [part] at (0, 800, 200) mm
      - 小方块（源对象） [part] at (0, 900, 200) mm
      - 小方块（源对象） [part] at (0, 0, 300) mm
      - 小方块（源对象） [part] at (0, 100, 300) mm
      - 小方块（源对象） [part] at (0, 200, 300) mm
      - 小方块（源对象） [part] at (0, 300, 300) mm
      - 小方块（源对象） [part] at (0, 400, 300) mm
      - 小方块（源对象） [part] at (0, 500, 300) mm
      - 小方块（源对象） [part] at (0, 600, 300) mm
      - 小方块（源对象） [part] at (0, 700, 300) mm
      - 小方块（源对象） [part] at (0, 800, 300) mm
      - 小方块（源对象） [part] at (0, 900, 300) mm
      - 小方块（源对象） [part] at (0, 0, 400) mm
      - 小方块（源对象） [part] at (0, 100, 400) mm
      - 小方块（源对象） [part] at (0, 200, 400) mm
      - 小方块（源对象） [part] at (0, 300, 400) mm
      - 小方块（源对象） [part] at (0, 400, 400) mm
      - 小方块（源对象） [part] at (0, 500, 400) mm
      - 小方块（源对象） [part] at (0, 600, 400) mm
      - 小方块（源对象） [part] at (0, 700, 400) mm
      - 小方块（源对象） [part] at (0, 800, 400) mm
      - 小方块（源对象） [part] at (0, 900, 400) mm
      - 小方块（源对象） [part] at (0, 0, 500) mm
      - 小方块（源对象） [part] at (0, 100, 500) mm
      - 小方块（源对象） [part] at (0, 200, 500) mm
      - 小方块（源对象） [part] at (0, 300, 500) mm
      - 小方块（源对象） [part] at (0, 400, 500) mm
      - 小方块（源对象） [part] at (0, 500, 500) mm
      - 小方块（源对象） [part] at (0, 600, 500) mm
      - 小方块（源对象） [part] at (0, 700, 500) mm
      - 小方块（源对象） [part] at (0, 800, 500) mm
      - 小方块（源对象） [part] at (0, 900, 500) mm
      - 小方块（源对象） [part] at (0, 0, 600) mm
      - 小方块（源对象） [part] at (0, 100, 600) mm
      - 小方块（源对象） [part] at (0, 200, 600) mm
      - 小方块（源对象） [part] at (0, 300, 600) mm
      - 小方块（源对象） [part] at (0, 400, 600) mm
      - 小方块（源对象） [part] at (0, 500, 600) mm
      - 小方块（源对象） [part] at (0, 600, 600) mm
      - 小方块（源对象） [part] at (0, 700, 600) mm
      - 小方块（源对象） [part] at (0, 800, 600) mm
      - 小方块（源对象） [part] at (0, 900, 600) mm
      - 小方块（源对象） [part] at (0, 0, 700) mm
      - 小方块（源对象） [part] at (0, 100, 700) mm
      - 小方块（源对象） [part] at (0, 200, 700) mm
      - 小方块（源对象） [part] at (0, 300, 700) mm
      - 小方块（源对象） [part] at (0, 400, 700) mm
      - 小方块（源对象） [part] at (0, 500, 700) mm
      - 小方块（源对象） [part] at (0, 600, 700) mm
      - 小方块（源对象） [part] at (0, 700, 700) mm
      - 小方块（源对象） [part] at (0, 800, 700) mm
      - 小方块（源对象） [part] at (0, 900, 700) mm
      - 小方块（源对象） [part] at (0, 0, 800) mm
      - 小方块（源对象） [part] at (0, 100, 800) mm
      - 小方块（源对象） [part] at (0, 200, 800) mm
      - 小方块（源对象） [part] at (0, 300, 800) mm
      - 小方块（源对象） [part] at (0, 400, 800) mm
      - 小方块（源对象） [part] at (0, 500, 800) mm
      - 小方块（源对象） [part] at (0, 600, 800) mm
      - 小方块（源对象） [part] at (0, 700, 800) mm
      - 小方块（源对象） [part] at (0, 800, 800) mm
      - 小方块（源对象） [part] at (0, 900, 800) mm
      - 小方块（源对象） [part] at (0, 0, 900) mm
      - 小方块（源对象） [part] at (0, 100, 900) mm
      - 小方块（源对象） [part] at (0, 200, 900) mm
      - 小方块（源对象） [part] at (0, 300, 900) mm
      - 小方块（源对象） [part] at (0, 400, 900) mm
      - 小方块（源对象） [part] at (0, 500, 900) mm
      - 小方块（源对象） [part] at (0, 600, 900) mm
      - 小方块（源对象） [part] at (0, 700, 900) mm
      - 小方块（源对象） [part] at (0, 800, 900) mm
      - 小方块（源对象） [part] at (0, 900, 900) mm
      - 小方块（源对象） [part] at (0, 0, 1000) mm
      - 小方块（源对象） [part] at (0, 100, 1000) mm
      - 小方块（源对象） [part] at (0, 200, 1000) mm
      - 小方块（源对象） [part] at (0, 300, 1000) mm
      - 小方块（源对象） [part] at (0, 400, 1000) mm
      - 小方块（源对象） [part] at (0, 500, 1000) mm
      - 小方块（源对象） [part] at (0, 600, 1000) mm
      - 小方块（源对象） [part] at (0, 700, 1000) mm
      - 小方块（源对象） [part] at (0, 800, 1000) mm
      - 小方块（源对象） [part] at (0, 900, 1000) mm
      - 小方块（源对象） [part] at (0, 0, 1100) mm
      - 小方块（源对象） [part] at (0, 100, 1100) mm
      - 小方块（源对象） [part] at (0, 200, 1100) mm
      - 小方块（源对象） [part] at (0, 300, 1100) mm
      - 小方块（源对象） [part] at (0, 400, 1100) mm
      - 小方块（源对象） [part] at (0, 500, 1100) mm
      - 小方块（源对象） [part] at (0, 600, 1100) mm
      - 小方块（源对象） [part] at (0, 700, 1100) mm
      - 小方块（源对象） [part] at (0, 800, 1100) mm
      - 小方块（源对象） [part] at (0, 900, 1100) mm
      - 小方块（源对象） [part] at (0, 0, 1200) mm
      - 小方块（源对象） [part] at (0, 100, 1200) mm
      - 小方块（源对象） [part] at (0, 200, 1200) mm
      - 小方块（源对象） [part] at (0, 300, 1200) mm
      - 小方块（源对象） [part] at (0, 400, 1200) mm
      - 小方块（源对象） [part] at (0, 500, 1200) mm
      - 小方块（源对象） [part] at (0, 600, 1200) mm
      - 小方块（源对象） [part] at (0, 700, 1200) mm
      - 小方块（源对象） [part] at (0, 800, 1200) mm
      - 小方块（源对象） [part] at (0, 900, 1200) mm
      - 小方块（源对象） [part] at (0, 0, 1300) mm
      - 小方块（源对象） [part] at (0, 100, 1300) mm
      - 小方块（源对象） [part] at (0, 200, 1300) mm
      - 小方块（源对象） [part] at (0, 300, 1300) mm
      - 小方块（源对象） [part] at (0, 400, 1300) mm
      - 小方块（源对象） [part] at (0, 500, 1300) mm
      - 小方块（源对象） [part] at (0, 600, 1300) mm
      - 小方块（源对象） [part] at (0, 700, 1300) mm
      - 小方块（源对象） [part] at (0, 800, 1300) mm
      - 小方块（源对象） [part] at (0, 900, 1300) mm
      - 小方块（源对象） [part] at (0, 0, 1400) mm
      - 小方块（源对象） [part] at (0, 100, 1400) mm
      - 小方块（源对象） [part] at (0, 200, 1400) mm
      - 小方块（源对象） [part] at (0, 300, 1400) mm
      - 小方块（源对象） [part] at (0, 400, 1400) mm
      - 小方块（源对象） [part] at (0, 500, 1400) mm
      - 小方块（源对象） [part] at (0, 600, 1400) mm
      - 小方块（源对象） [part] at (0, 700, 1400) mm
      - 小方块（源对象） [part] at (0, 800, 1400) mm
      - 小方块（源对象） [part] at (0, 900, 1400) mm
      - 小方块（源对象） [part] at (0, 0, 1500) mm
      - 小方块（源对象） [part] at (0, 100, 1500) mm
      - 小方块（源对象） [part] at (0, 200, 1500) mm
      - 小方块（源对象） [part] at (0, 300, 1500) mm
      - 小方块（源对象） [part] at (0, 400, 1500) mm
      - 小方块（源对象） [part] at (0, 500, 1500) mm
      - 小方块（源对象） [part] at (0, 600, 1500) mm
      - 小方块（源对象） [part] at (0, 700, 1500) mm
      - 小方块（源对象） [part] at (0, 800, 1500) mm
      - 小方块（源对象） [part] at (0, 900, 1500) mm
      - 小方块（源对象） [part] at (0, 0, 1600) mm
      - 小方块（源对象） [part] at (0, 100, 1600) mm
      - 小方块（源对象） [part] at (0, 200, 1600) mm
      - 小方块（源对象） [part] at (0, 300, 1600) mm
      - 小方块（源对象） [part] at (0, 400, 1600) mm
      - 小方块（源对象） [part] at (0, 500, 1600) mm
      - 小方块（源对象） [part] at (0, 600, 1600) mm
      - 小方块（源对象） [part] at (0, 700, 1600) mm
      - 小方块（源对象） [part] at (0, 800, 1600) mm
      - 小方块（源对象） [part] at (0, 900, 1600) mm
      - 小方块（源对象） [part] at (0, 0, 1700) mm
      - 小方块（源对象） [part] at (0, 100, 1700) mm
      - 小方块（源对象） [part] at (0, 200, 1700) mm
      - 小方块（源对象） [part] at (0, 300, 1700) mm
      - 小方块（源对象） [part] at (0, 400, 1700) mm
      - 小方块（源对象） [part] at (0, 500, 1700) mm
      - 小方块（源对象） [part] at (0, 600, 1700) mm
      - 小方块（源对象） [part] at (0, 700, 1700) mm
      - 小方块（源对象） [part] at (0, 800, 1700) mm
      - 小方块（源对象） [part] at (0, 900, 1700) mm
      - 小方块（源对象） [part] at (0, 0, 1800) mm
      - 小方块（源对象） [part] at (0, 100, 1800) mm
      - 小方块（源对象） [part] at (0, 200, 1800) mm
      - 小方块（源对象） [part] at (0, 300, 1800) mm
      - 小方块（源对象） [part] at (0, 400, 1800) mm
      - 小方块（源对象） [part] at (0, 500, 1800) mm
      - 小方块（源对象） [part] at (0, 600, 1800) mm
      - 小方块（源对象） [part] at (0, 700, 1800) mm
      - 小方块（源对象） [part] at (0, 800, 1800) mm
      - 小方块（源对象） [part] at (0, 900, 1800) mm
      - 小方块（源对象） [part] at (0, 0, 1900) mm
      - 小方块（源对象） [part] at (0, 100, 1900) mm
      - 小方块（源对象） [part] at (0, 200, 1900) mm
      - 小方块（源对象） [part] at (0, 300, 1900) mm
      - 小方块（源对象） [part] at (0, 400, 1900) mm
      - 小方块（源对象） [part] at (0, 500, 1900) mm
      - 小方块（源对象） [part] at (0, 600, 1900) mm
      - 小方块（源对象） [part] at (0, 700, 1900) mm
      - 小方块（源对象） [part] at (0, 800, 1900) mm
      - 小方块（源对象） [part] at (0, 900, 1900) mm
    - 小方块（源对象） [part]
  - 俄罗斯方块随机生成器 [smart component]
      properties: Random_TetrisID=0; Brick=(none)
      signals: DI NewBrick
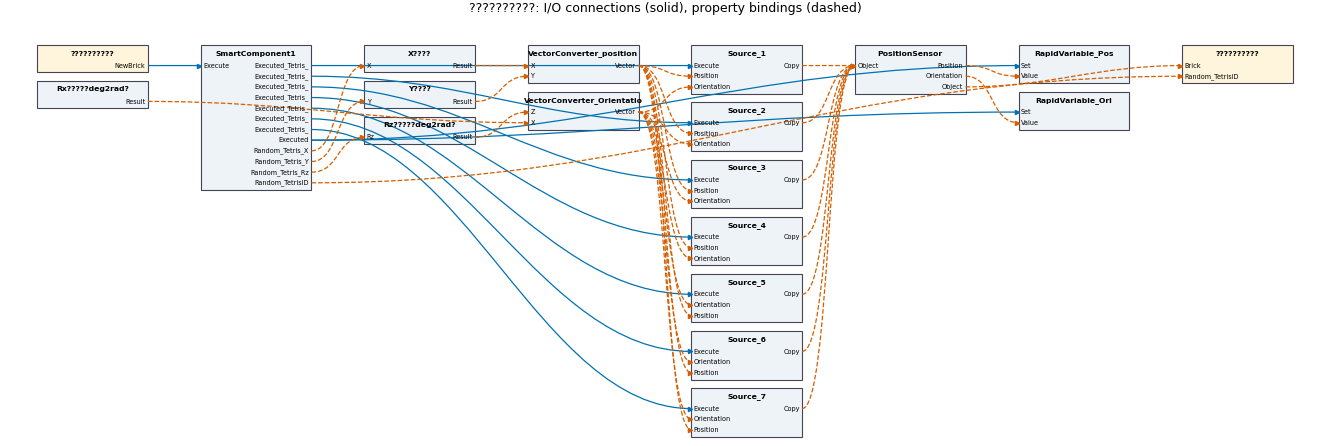
      connections:
        SmartComponent1.Executed_Tetris_1 -> Source_1.Execute
        SmartComponent1.Executed_Tetris_2 -> Source_2.Execute
        SmartComponent1.Executed_Tetris_3 -> Source_3.Execute
        SmartComponent1.Executed_Tetris_4 -> Source_4.Execute
        SmartComponent1.Executed_Tetris_5 -> Source_5.Execute
        SmartComponent1.Executed_Tetris_6 -> Source_6.Execute
        SmartComponent1.Executed_Tetris_7 -> Source_7.Execute
        SmartComponent1.Executed -> RapidVariable_Pos.Set
        SmartComponent1.Executed -> RapidVariable_Ori.Set
        俄罗斯方块随机生成器.NewBrick -> SmartComponent1.Execute
        X单位转化.Result => VectorConverter_position.X
        Y单位转化.Result => VectorConverter_position.Y
        Rz单位转化（deg2rad）.Result => VectorConverter_Orientation.Z
        Source_1.Copy => PositionSensor.Object
        Source_4.Copy => PositionSensor.Object
        Source_7.Copy => PositionSensor.Object
        Source_5.Copy => PositionSensor.Object
        Source_2.Copy => PositionSensor.Object
        Source_3.Copy => PositionSensor.Object
        Source_6.Copy => PositionSensor.Object
        VectorConverter_position.Vector => Source_1.Position
        VectorConverter_position.Vector => Source_2.Position
        VectorConverter_position.Vector => Source_3.Position
        VectorConverter_position.Vector => Source_4.Position
        VectorConverter_Orientation.Vector => Source_3.Orientation
        VectorConverter_Orientation.Vector => Source_6.Orientation
        VectorConverter_Orientation.Vector => Source_1.Orientation
        VectorConverter_Orientation.Vector => Source_4.Orientation
        VectorConverter_Orientation.Vector => Source_5.Orientation
        VectorConverter_Orientation.Vector => Source_2.Orientation
        VectorConverter_position.Vector => Source_5.Position
        VectorConverter_position.Vector => Source_6.Position
        VectorConverter_Orientation.Vector => Source_7.Orientation
        VectorConverter_position.Vector => Source_7.Position
        PositionSensor.Position => RapidVariable_Pos.Value
        PositionSensor.Orientation => RapidVariable_Ori.Value
        PositionSensor.Object => 俄罗斯方块随机生成器.Brick
        Rx单位转化（deg2rad）.Result => VectorConverter_Orientation.X
        SmartComponent1.Random_Tetris_X => X单位转化.X
        SmartComponent1.Random_Tetris_Y => Y单位转化.Y
        SmartComponent1.Random_Tetris_Rz => Rz单位转化（deg2rad）.Rz
        SmartComponent1.Random_TetrisID => 俄罗斯方块随机生成器.Random_TetrisID
    - VectorConverter_Orientation [smart component, from Components\VectorConverter.rslib]
        properties: X=-1.5707963267949; Y=0; Z=0; Vector=[-1.5707963267949 0 0]
    - VectorConverter_position [smart component, from Components\VectorConverter.rslib]
        properties: X=0; Y=0; Z=0.1; Vector=[0 0 0.1]
    - 俄罗斯方块组1 [graphiccomponentgroup] at (0, 0, 100) mm, rotated rx -90 ry 0 rz 0 deg
      - 俄罗斯方块单元1_1 [part]
      - 俄罗斯方块单元1_4 [part] at (100, 0, 200) mm
      - 俄罗斯方块单元1_2 [part] at (0, 0, 100) mm
      - 俄罗斯方块单元1_3 [part] at (0, 0, 200) mm
    - Source_1 [smart component, from Components\Source.rslib]
        properties: Source=俄罗斯方块组1; Copy=(none); Parent=俄罗斯方块随机生成器; Position=[0 0 0.1]; Orientation=[-1.5707963267949 0 0]; Transient=true; PhysicsBehavior=0
    - 俄罗斯方块组2 [graphiccomponentgroup] at (0, 0, 100) mm, rotated rx -90 ry 0 rz 0 deg
      - 俄罗斯方块单元2_4 [part] at (100, 0, 200) mm
      - 俄罗斯方块单元2_1 [part]
      - 俄罗斯方块单元2_2 [part] at (0, 0, 100) mm
      - 俄罗斯方块单元2_3 [part] at (100, 0, 100) mm
    - 俄罗斯方块组5 [graphiccomponentgroup] at (0, 0, 100) mm, rotated rx -90 ry 0 rz 0 deg
      - 俄罗斯方块单元5_1 [part]
      - 俄罗斯方块单元5_2 [part] at (100, 0, 0) mm
      - 俄罗斯方块单元5_3 [part] at (200, 0, 0) mm
      - 俄罗斯方块单元5_4 [part] at (300, 0, 0) mm
      - 吸盘 [smart component] at (-54.41, 502.5, 1697.5) mm, rotated rx 180 ry 60 rz 0 deg
          signals: DI Grab, DO Delete_Row
          connections:
            吸盘.Grab -> LineSensor.Active
            吸盘.Grab -> LogicGate.InputA
            LogicGate.Output -> Detacher.Execute
            Detacher.Executed -> 吸盘.Delete_Row
            吸盘.Grab -> LineSensor.Active
            LineSensor.SensorOut -> Attacher.Execute
            Attacher.Child => Detacher.Child
            LineSensor.SensedPart => Attacher.Child
        - LogicGate [smart component, from Components\LogicGate.rslib]
            properties: Operator=NOT; Delay=0
        - Attacher [smart component, from Components\Attacher.rslib]
            properties: Parent=吸盘; Flange=0; Child=(none); Mount=false; Offset=[0 0 0]; Orientation=[0 0 0]
        - Detacher [smart component, from Components\Detacher.rslib]
            properties: Child=(none); KeepPosition=true
        - LineSensor [smart component, from Components\LineSensor.rslib] at (-173.21, 0, -100) mm
            properties: Start=[0.0150000000000043 0.0185000000000005 0.0375000000000047]; End=[0.115000000000004 0.0185000000000005 0.0375000000000047]; Radius=0.003; SensedPart=(none); SensedPoint=[-0.0731893844604492 0.484 1.65502087402344]
          - _sensorPart_ [part]
    - 俄罗斯方块组4 [graphiccomponentgroup] at (0, 0, 100) mm, rotated rx -90 ry 0 rz 0 deg
      - 俄罗斯方块单元4_1 [part] at (0, 0, 100) mm
      - 俄罗斯方块单元4_2 [part]
      - 俄罗斯方块单元4_3 [part] at (-100, 0, 100) mm
      - 俄罗斯方块单元4_4 [part] at (-100, 0, 200) mm
    - 俄罗斯方块组3 [graphiccomponentgroup] at (0, 0, 100) mm, rotated rx -90 ry 0 rz 0 deg
      - 俄罗斯方块单元3_1 [part]
      - 俄罗斯方块单元3_2 [part] at (0, 0, 100) mm
      - 俄罗斯方块单元3_3 [part] at (0, 0, 200) mm
      - 俄罗斯方块单元3_4 [part] at (-100, 0, 200) mm
    - 俄罗斯方块组6 [graphiccomponentgroup] at (0, 0, 100) mm, rotated rx -90 ry 0 rz 0 deg
      - 俄罗斯方块单元6_1 [part] at (0, 0, 100) mm
      - 俄罗斯方块单元6_2 [part]
      - 俄罗斯方块单元6_3 [part] at (100, 0, 100) mm
      - 俄罗斯方块单元6_4 [part] at (100, 0, 0) mm
    - 俄罗斯方块组7 [graphiccomponentgroup] at (0, 0, 100) mm, rotated rx -90 ry 0 rz 0 deg
      - 俄罗斯方块单元7_4 [part] at (100, 0, 100) mm
      - 俄罗斯方块单元7_1 [part]
      - 俄罗斯方块单元7_2 [part] at (100, 0, 0) mm
      - 俄罗斯方块单元7_3 [part] at (200, 0, 0) mm
    - Source_2 [smart component, from Components\Source.rslib]
        properties: Source=俄罗斯方块组2; Copy=(none); Parent=俄罗斯方块随机生成器; Position=[0 0 0.1]; Orientation=[-1.5707963267949 0 0]; Transient=true; PhysicsBehavior=0
    - Source_3 [smart component, from Components\Source.rslib]
        properties: Source=俄罗斯方块组3; Copy=(none); Parent=俄罗斯方块随机生成器; Position=[0 0 0.1]; Orientation=[-1.5707963267949 0 0]; Transient=true; PhysicsBehavior=0
    - Source_4 [smart component, from Components\Source.rslib]
        properties: Source=俄罗斯方块组4; Copy=(none); Parent=俄罗斯方块随机生成器; Position=[0 0 0.1]; Orientation=[-1.5707963267949 0 0]; Transient=true; PhysicsBehavior=0
    - Source_5 [smart component, from Components\Source.rslib]
        properties: Source=俄罗斯方块组5; Copy=(none); Parent=俄罗斯方块随机生成器; Position=[0 0 0.1]; Orientation=[-1.5707963267949 0 0]; Transient=true; PhysicsBehavior=0
    - Source_6 [smart component, from Components\Source.rslib]
        properties: Source=俄罗斯方块组6; Copy=(none); Parent=俄罗斯方块随机生成器; Position=[0 0 0.1]; Orientation=[-1.5707963267949 0 0]; Transient=true; PhysicsBehavior=0
    - Source_7 [smart component, from Components\Source.rslib]
        properties: Source=俄罗斯方块组7; Copy=(none); Parent=俄罗斯方块随机生成器; Position=[0 0 0.1]; Orientation=[-1.5707963267949 0 0]; Transient=true; PhysicsBehavior=0
    - X单位转化 [smart component, from Components\Expression.rslib]
        properties: Expression=X/1000; Result=0; X=0
    - Y单位转化 [smart component, from Components\Expression.rslib]
        properties: Expression=Y/1000; Result=0; Y=0
    - Rz单位转化（deg2rad） [smart component, from Components\Expression.rslib]
        properties: Expression=Rz*PI/180; Result=0; Y=0; Rz=0
    - PositionSensor [smart component, from Components\PositionSensor.rslib]
        properties: Object=(none); Reference=Object; ReferenceObject=IRB2600_12_165_C_01_2; Position=[0.330000009141263 0.875000006811872 0.0999999498724324]; Orientation=[0 1.5707963267949 -3.92971923814893E-08]
    - RapidVariable_Pos [smart component, from Components\RapidVariable.rslib]
        properties: DataType=pos; Controller=Controller_IRB2600_12_165_C; Task=T_ROB1; Module=Module1; Variable=T_Pos; Value=[0.330000009141263 0.875000006811872 0.0999999498724324]
    - RapidVariable_Ori [smart component, from Components\RapidVariable.rslib]
        properties: DataType=orient; Controller=Controller_IRB2600_12_165_C; Task=T_ROB1; Module=Module1; Variable=T_Ori; Value=[0 1.5707963267949 -3.92971923814893E-08]
    - Rx单位转化（deg2rad） [smart component, from Components\Expression.rslib]
        properties: Expression=-PI/2; Result=-1.5707963267949; Y=0; Rz=28.2352941176471
    - SmartComponent1 [smart component]
        properties: Random_Tetris_X=0; Random_Tetris_Y=0; Random_Tetris_Rz=0; Random_TetrisID=0
        signals: DI Execute, DO Executed, DO Executed_Tetris_1, DO Executed_Tetris_2, DO Executed_Tetris_3, DO Executed_Tetris_4, DO Executed_Tetris_5, DO Executed_Tetris_6, DO Executed_Tetris_7
  - 俄罗斯方块AI算法（基于PD算法） [smart component]
      properties: Random_TetrisID=0; Tetris_AI_y=0; Tetris_AI_z=0; Tetris_AI_Rx_Times=0; GameOver=0; Brick=(none); InPosition=0
      signals: DI NewGame, DI NewBrick, DO GameOver, DI AI_No_Fill_In, DI AI_Fill_In
      connections:
        俄罗斯方块AI算法（基于PD算法）.NewGame -> MultiTimer.Reset
        俄罗斯方块AI算法（基于PD算法）.NewGame -> LogicSRLatch.Reset
        MultiTimer.Output1 -> LogicSRLatch.Set
        LogicSRLatch.Output -> 俄罗斯方块AI算法（基于PD算法）.GameOver
        俄罗斯方块AI算法（基于PD算法）.NewGame -> TetrisAI.NewGame
        俄罗斯方块AI算法（基于PD算法）.AI_No_Fill_In -> TetrisAI.AI_PD_No_Fill_In
        俄罗斯方块AI算法（基于PD算法）.AI_Fill_In -> TetrisAI.AI_PD_Fill_In
        俄罗斯方块AI算法（基于PD算法）.NewBrick -> TetrisAI.NewBrick
        TetrisAI.Executed -> RapidVariable.Set
        TetrisAI.Executed -> RapidVariable_2.Set
        TetrisAI.Executed -> RapidVariable_3.Set
        俄罗斯方块AI算法（基于PD算法）.Random_TetrisID => TetrisAI.Random_TetrisID
        TetrisAI.Tetris_AI_x => RapidVariable.Value
        TetrisAI.Tetris_AI_y => RapidVariable_2.Value
        TetrisAI.Tetris_AI_Rz_Times => RapidVariable_3.Value
        TetrisAI.GameOver => 俄罗斯方块AI算法（基于PD算法）.GameOver
    - RapidVariable [smart component, from Components\RapidVariable.rslib]
        properties: DataType=num; Controller=Controller_IRB2600_12_165_C; Task=T_ROB1; Module=Module1; Variable=AI_y; Value=0
    - RapidVariable_2 [smart component, from Components\RapidVariable.rslib]
        properties: DataType=num; Controller=Controller_IRB2600_12_165_C; Task=T_ROB1; Module=Module1; Variable=AI_z; Value=0
    - RapidVariable_3 [smart component, from Components\RapidVariable.rslib]
        properties: DataType=num; Controller=Controller_IRB2600_12_165_C; Task=T_ROB1; Module=Module1; Variable=AI_Rx_T_times; Value=0
    - LogicSRLatch [smart component, from Components\LogicSRLatch.rslib]
    - MultiTimer [smart component, from Components\MultiTimer.rslib]
        properties: Count=1; CurrentTime=0; Time1=600
    - TetrisAI [smart component]
        properties: Random_TetrisID=0; Tetris_AI_x=800; Tetris_AI_y=200; Tetris_AI_Rz_Times=2; GameOver=0
        signals: DI NewGame, DI AI_PD_Fill_In, DI AI_PD_No_Fill_In, DI NewBrick, DO Executed
  - 气动吸盘 [smart component]
      properties: Brick=(none)
      signals: DI Attach_Brick
      connections:
        LogicGate_2.Output -> Detacher.Execute
        气动吸盘.Attach_Brick -> LineSensor.Active
        LineSensor.SensorOut -> Attacher.Execute
        气动吸盘.Attach_Brick -> LogicGate_2.InputA
        气动吸盘.Brick => Attacher.Child
        气动吸盘.Brick => Detacher.Child
    - Attacher [smart component, from Components\Attacher.rslib]
        properties: Parent=My_Mechanism_Vacuum; Flange=0; Child=(none); Mount=false; Offset=[0 0 0]; Orientation=[0 0 0]
    - Detacher [smart component, from Components\Detacher.rslib]
        properties: Child=(none); KeepPosition=true
    - LineSensor [smart component, from Components\LineSensor.rslib] at (1280, -193.92, 1283.49) mm, rotated rx -60 ry 0 rz 0 deg
        properties: Start=[1.11022302462516E-16 0 -0.0465000000000002]; End=[1.11022302462516E-16 0 0.0234999999999999]; Radius=0.003; SensedPart=(none); SensedPoint=[0 0 0]
      - _sensorPart_ [part]
    - LogicGate_2 [smart component, from Components\LogicGate.rslib]
        properties: Operator=NOT; Delay=0
  - IRB2600_12_165_C_01_2 [mechanism, from Robots\IRB2600_12_165_C_01.rslib] at (1280, 730, 300) mm, rotated rx 0 ry 0 rz -90 deg; joint values [0, 0, 0, 0, 0.5236, 0] (rad or m)
  - 机器人吸盘外轴 [smart component]
      signals: DI AI_Rx_T_times_1, DI AI_Rx_T_times_2, DI AI_Rx_T_times_3, DI AI_Rx_T_times_4
      connections:
        机器人吸盘外轴.AI_Rx_T_times_1 -> PoseMover_1.Execute
        机器人吸盘外轴.AI_Rx_T_times_2 -> PoseMover_2.Execute
        机器人吸盘外轴.AI_Rx_T_times_3 -> PoseMover_3.Execute
        机器人吸盘外轴.AI_Rx_T_times_4 -> PoseMover_4.Execute
    - PoseMover_1 [smart component, from Components\PoseMover.rslib]
        properties: Mechanism=My_Mechanism_Vacuum; Pose=2; Duration=0.5
    - PoseMover_3 [smart component, from Components\PoseMover.rslib]
        properties: Mechanism=My_Mechanism_Vacuum; Pose=4; Duration=0.5
    - PoseMover_4 [smart component, from Components\PoseMover.rslib]
        properties: Mechanism=My_Mechanism_Vacuum; Pose=0; Duration=0.5
    - PoseMover_2 [smart component, from Components\PoseMover.rslib]
        properties: Mechanism=My_Mechanism_Vacuum; Pose=3; Duration=0.5
  - My_Mechanism_Vacuum [mechanism, from Libraries\My_Mechanism_Vacuum.rslib] at (1280, -288.61, 1517.5) mm, rotated rx -60 ry 0 rz 0 deg; joint values [0] (rad or m)
  - 底座 [part] at (1280, 730, 0) mm
  - UCS [frame] at (1507.5, 502.5, 0) mm
Attachment: 满行检测与下坠_1 is attached to 扫描式传感器 / L1
Attachment: 满行检测与下坠_2 is attached to 扫描式传感器 / L1
Attachment: 满行检测与下坠_3 is attached to 扫描式传感器 / L1
Attachment: 满行检测与下坠_4 is attached to 扫描式传感器 / L1
Attachment: 满行检测与下坠_5 is attached to 扫描式传感器 / L1
Attachment: 满行检测与下坠_6 is attached to 扫描式传感器 / L1
Attachment: 满行检测与下坠_7 is attached to 扫描式传感器 / L1
Attachment: 满行检测与下坠_8 is attached to 扫描式传感器 / L1
Attachment: 满行检测与下坠_9 is attached to 扫描式传感器 / L1
Attachment: 满行检测与下坠_10 is attached to 扫描式传感器 / L1
Attachment: 满行检测与下坠_11 is attached to 扫描式传感器 / L1
Attachment: 满行检测与下坠_12 is attached to 扫描式传感器 / L1
Attachment: 满行检测与下坠_13 is attached to 扫描式传感器 / L1
Attachment: 满行检测与下坠_14 is attached to 扫描式传感器 / L1
Attachment: 满行检测与下坠_15 is attached to 扫描式传感器 / L1
Attachment: 满行检测与下坠_16 is attached to 扫描式传感器 / L1
Attachment: 满行检测与下坠_17 is attached to 扫描式传感器 / L1
Attachment: 满行检测与下坠_18 is attached to 扫描式传感器 / L1
Attachment: 满行检测与下坠_19 is attached to 扫描式传感器 / L1
Attachment: 满行检测与下坠_20 is attached to 扫描式传感器 / L1
Attachment: LineSensor is attached to My_Mechanism_Vacuum / L2
Attachment: My_Mechanism_Vacuum is attached to IRB2600_12_165_C_01_2 / Link6
Station logic (signal -> signal, property => property):
  吸盘.Delete_Row -> 删行控制器.Rows_Delete
  俄罗斯方块AI算法（基于PD算法）.GameOver -> Controller_IRB2600_12_165_C.GameOver0
  Controller_IRB2600_12_165_C.NewGame0 -> 俄罗斯方块AI算法（基于PD算法）.NewGame
  Controller_IRB2600_12_165_C.NewBrick0 -> 俄罗斯方块随机生成器.NewBrick
  Controller_IRB2600_12_165_C.Attach_Block0 -> 气动吸盘.Attach_Brick
  Controller_IRB2600_12_165_C.Rows_Delete0 -> 删行控制器.Rows_Delete
  Controller_IRB2600_12_165_C.AI_Rx_T_times_10 -> 机器人吸盘外轴.AI_Rx_T_times_1
  Controller_IRB2600_12_165_C.AI_Rx_T_times_20 -> 机器人吸盘外轴.AI_Rx_T_times_2
  Controller_IRB2600_12_165_C.AI_Rx_T_times_30 -> 机器人吸盘外轴.AI_Rx_T_times_3
  Controller_IRB2600_12_165_C.AI_Rx_T_times_40 -> 机器人吸盘外轴.AI_Rx_T_times_4
  Controller_IRB2600_12_165_C.NewBrick0 -> 俄罗斯方块AI算法（基于PD算法）.NewBrick
  Controller_IRB2600_12_165_C.AI_Fill_In0 -> 俄罗斯方块AI算法（基于PD算法）.AI_Fill_In
  Controller_IRB2600_12_165_C.AI_No_Fill_In0 -> 俄罗斯方块AI算法（基于PD算法）.AI_No_Fill_In
  俄罗斯方块随机生成器.Brick => 气动吸盘.Brick
  俄罗斯方块随机生成器.Random_TetrisID => 俄罗斯方块AI算法（基于PD算法）.Random_TetrisID

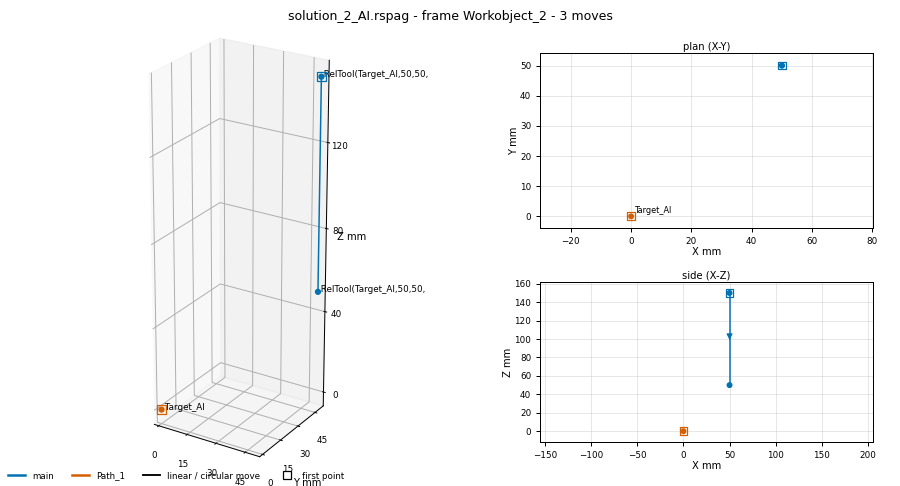
[picture p0: tool path of solution_2_AI.rspag in frame Workobject_2, 3 of 10 moves have a stored position in this frame; points joined in program order, loops and branches not executed]
--- Backups/Controller_IRB2600_12_165_C/RAPID/TASK1/PROGMOD/Module1.mod ---
MODULE Module1
    VAR num ID:=1;
    VAR num AI_y:=0;
    VAR num AI_z:=0;
    VAR num AI_Rx_T_times:=0;
    VAR pose T_Pose;
    VAR pos T_Pos;
    VAR orient T_Ori;
    VAR pos W1_Pos;
    VAR pos W2_Pos;
    VAR pos AI_Pos;

    CONST robtarget Brick:=[[50,0,50],[0.707106781,0.707106781,0,0],[-1,0,1,0],[9E+09,9E+09,9E+09,9E+09,9E+09,9E+09]];
    CONST robtarget Target_Process:=[[680,630,150],[0.707106781,0.707106781,0,0],[0,-1,-1,1],[9E+09,9E+09,9E+09,9E+09,9E+09,9E+09]];
    CONST robtarget Target_AI:=[[0,0,0],[1,0,0,0],[1,0,0,1],[9E+09,9E+09,9E+09,9E+09,9E+09,9E+09]];

    PERS wobjdata Workobject_1:=[FALSE,TRUE,"",[[36.2745,-840.392,-200],[0.0370071,-0.0370071,0.706138,-0.706138]],[[0,0,0],[1,0,0,0]]];
    PERS wobjdata Workobject_2:=[FALSE,TRUE,"",[[-170,780,-200],[0.707107,0.707107,0,0]],[[0,0,0],[1,0,0,0]]];
    PERS tooldata ToolFrame:=[TRUE,[[250,0,35],[0,-0.707107,0.707107,0]],[1,[0,1,0],[1,0,0,0],0,0,0]];

    PROC main()
        MoveAbsJ [[0,0,0,0,30,0],[9E+09,9E+09,9E+09,9E+09,9E+09,9E+09]],v7000,fine,tool0;
        SetDO NewGame0,0;
        SetDO NewGame0,1;
        !SetDO AI_No_Fill_In0,1;//AI_No_Fill_In0 and SetDo AI_Fill_In0 only can choice one.
        SetDo AI_Fill_In0,1;
        WaitTime 0.2;
        WHILE GameOver0<>1 DO
            Workobject_1.uframe.trans:=[730,-1280,-200];
            Workobject_2.uframe.trans:=[-270,780,-300];
            W2_Pos:=Workobject_2.uframe.trans;
            PulseDO NewBrick0;
            WaitTime 0.1;
            T_Pose:=[T_Pos,T_Ori];
            Workobject_1.uframe:=T_Pose;
            AI_Pos:=W2_Pos+[AI_y,0,AI_z];
            Workobject_2.uframe.trans:=AI_Pos;
            MoveJ Brick,v7000,fine,ToolFrame\WObj:=Workobject_1;
            SetDO Attach_Block0,1;
            W1_Pos:=Workobject_1.uframe.trans;
            IF W1_Pos.y>=-700 THEN
                W1_Pos.y:=-700;
                MoveJ Brick,v7000,z200,ToolFrame\WObj:=Workobject_1;
            ENDIF
            MoveJ RelTool(Brick,0,0,200),v7000,z200,ToolFrame\WObj:=Workobject_1;
            MoveJ Target_Process,v7000,z200,ToolFrame\WObj:=wobj0;
            IF AI_Rx_T_times=1 THEN
                PulseDO AI_Rx_T_times_10;
            ELSEIF AI_Rx_T_times=2 THEN
                PulseDO AI_Rx_T_times_20;
            ELSEIF AI_Rx_T_times=3 THEN
                PulseDO AI_Rx_T_times_30;
            ELSEIF AI_Rx_T_times=4 THEN
                PulseDO AI_Rx_T_times_40;
            ENDIF
            MoveL RelTool(Target_AI,50,50,150),v7000,z200,ToolFrame\WObj:=Workobject_2;
            MoveL RelTool(Target_AI,50,50,50),v7000,fine,ToolFrame\WObj:=Workobject_2;
            SetDO Attach_Block0,0;
            WaitTime 0.1;
            PulseDO Rows_Delete0;
            PulseDO AI_Rx_T_times_40;
            WaitTime 0.1;
        ENDWHILE
    ENDPROC

    PROC Path_1()
        MoveL Brick,v1000,z100,ToolFrame\WObj:=Workobject_1;
        MoveL Target_Process,v1000,z100,ToolFrame\WObj:=wobj0;
        MoveL Target_AI,v1000,z100,tool0\WObj:=Workobject_2;
    ENDPROC
ENDMODULE

--- Backups/Controller_IRB2600_12_165_C/SYSPAR/EIO.cfg ---
EIO:CFG_1.0:6:1::
#
EIO_SIGNAL:

      -Name "NewGame0" -SignalType "DO"

      -Name "GameOver0" -SignalType "DI"

      -Name "NewBrick0" -SignalType "DO"

      -Name "Attach_Block0" -SignalType "DO"

      -Name "Rows_Delete0" -SignalType "DO"

      -Name "AI_Rx_T_times_10" -SignalType "DO"

      -Name "AI_Rx_T_times_20" -SignalType "DO"

      -Name "AI_Rx_T_times_30" -SignalType "DO"

      -Name "AI_Rx_T_times_40" -SignalType "DO"

      -Name "AI_Fill_In0" -SignalType "DO"

      -Name "AI_No_Fill_In0" -SignalType "DO"
